LIN {X 0,Y 302.837,Z 619.691,A -85,B 0,C 180,E1 -24110.683,E2 -24110.683} C_VEL
LIN {X 0,Y 303.085,Z 619.66,A -85,B 0,C 180,E1 -24113.589,E2 -24113.589} C_VEL
LIN {X 0,Y 303.031,Z 619.668,A -85,B 0,C 180,E1 -24117.351,E2 -24117.351} C_VEL
LIN {X 0,Y 303.108,Z 619.662,A -85,B 0,C 180,E1 -24120,E2 -24120} C_VEL
LIN {X 0,Y 303.072,Z 619.665,A -85,B 0,C 180,E1 -24123.976,E2 -24123.976} C_VEL
LIN {X 0,Y 302.989,Z 619.674,A -85,B 0,C 180,E1 -24126.638,E2 -24126.638} C_VEL
LIN {X 0,Y 302.772,Z 619.699,A -85,B 0,C 180,E1 -24130.666,E2 -24130.666} C_VEL
LIN {X 0,Y 302.721,Z 619.706,A -85,B 0,C 180,E1 -24133.638,E2 -24133.638} C_VEL
LIN {X 0,Y 302.599,Z 619.723,A -85,B 0,C 180,E1 -24137.513,E2 -24137.513} C_VEL
LIN {X 0,Y 302.618,Z 619.72,A -85,B 0,C 180,E1 -24141.737,E2 -24141.737} C_VEL
LIN {X 0,Y 302.58,Z 619.729,A -85,B 0,C 180,E1 -24146.094,E2 -24146.094} C_VEL
LIN {X 0,Y 302.525,Z 619.73,A -85,B 0,C 180,E1 -24149.093,E2 -24149.093} C_VEL
LIN {X 0,Y 302.517,Z 619.734,A -85,B 0,C 180,E1 -24152.178,E2 -24152.178} C_VEL
LIN {X 0,Y 302.558,Z 619.731,A -85,B 0,C 180,E1 -24155.877,E2 -24155.877} C_VEL
LIN {X 0,Y 302.508,Z 619.732,A -85,B 0,C 180,E1 -24158.695,E2 -24158.695} C_VEL
LIN {X 0,Y 302.518,Z 619.734,A -85,B 0,C 180,E1 -24162.19,E2 -24162.19} C_VEL
LIN {X 0,Y 302.516,Z 619.736,A -85,B 0,C 180,E1 -24165.84,E2 -24165.84} C_VEL
LIN {X 0,Y 301.902,Z 619.818,A -85,B 0,C 180,E1 -24166.951,E2 -24166.951} C_VEL
LIN {X 0,Y 299.026,Z 620.17,A -85,B 0,C 180,E1 -24168.76,E2 -24168.76} C_VEL
LIN {X 0,Y 296.57,Z 620.472,A -85,B 0,C 180,E1 -24170.228,E2 -24170.228} C_VEL
LIN {X 0,Y 295.543,Z 620.598,A -85,B 0,C 180,E1 -24171.366,E2 -24171.366} C_VEL
LIN {X 0,Y 295.477,Z 620.608,A -85,B 0,C 180,E1 -24171.752,E2 -24171.752} C_VEL
LIN {X 0,Y 295.463,Z 620.611,A -85,B 0,C 180,E1 -24175.323,E2 -24175.323} C_VEL
LIN {X 0,Y 295.472,Z 620.609,A -85,B 0,C 180,E1 -24178.585,E2 -24178.585} C_VEL
LIN {X 0,Y 295.688,Z 620.648,A -85,B 0,C 180,E1 -24182.966,E2 -24182.966} C_VEL
LIN {X 0,Y 297.523,Z 631.227,A -85,B 0,C 180,E1 -24186.408,E2 -24186.408} C_VEL
LIN {X 0,Y 296.857,Z 636.884,A -85,B 0,C 180,E1 -24188.184,E2 -24188.184} C_VEL
LIN {X 0,Y 296.097,Z 642.614,A -85,B 0,C 180,E1 -24189.913,E2 -24189.913} C_VEL
LIN {X 0,Y 297.168,Z 664.042,A -85,B 0,C 180,E1 -24190.732,E2 -24190.732} C_VEL
LIN {X 0,Y 299.254,Z 687.174,A -85,B 0,C 180,E1 -24191.624,E2 -24191.624} C_VEL
LIN {X 0,Y 297.458,Z 748.577,A -85,B 0,C 180,E1 -24193.894,E2 -24193.894} C_VEL
LIN {X 0,Y 296.972,Z 759.313,A -85,B 0,C 180,E1 -24194.438,E2 -24194.438} C_VEL
LIN {X 0,Y 296.571,Z 769.561,A -85,B 0,C 180,E1 -24195.123,E2 -24195.123} C_VEL
LIN {X 0,Y 296.15,Z 779.319,A -85,B 0,C 180,E1 -24195.942,E2 -24195.942} C_VEL
LIN {X 0,Y 295.546,Z 789.452,A -85,B 0,C 180,E1 -24196.989,E2 -24196.989} C_VEL
LIN {X 0,Y 294.854,Z 798.937,A -85,B 0,C 180,E1 -24198.177,E2 -24198.177} C_VEL
LIN {X 0,Y 294.346,Z 806.961,A -85,B 0,C 180,E1 -24199.373,E2 -24199.373} C_VEL
LIN {X 0,Y 293.912,Z 814.791,A -85,B 0,C 180,E1 -24200.743,E2 -24200.743} C_VEL
LIN {X 0,Y 293.521,Z 822.971,A -85,B 0,C 180,E1 -24202.458,E2 -24202.458} C_VEL
LIN {X 0,Y 293.293,Z 829.787,A -85,B 0,C 180,E1 -24204.175,E2 -24204.175} C_VEL
LIN {X 0,Y 293.161,Z 835.457,A -85,B 0,C 180,E1 -24205.89,E2 -24205.89} C_VEL
LIN {X 0,Y 293.07,Z 839.33,A -85,B 0,C 180,E1 -24207.26,E2 -24207.26} C_VEL
LIN {X 0,Y 292.986,Z 843.949,A -85,B 0,C 180,E1 -24209.315,E2 -24209.315} C_VEL
LIN {X 0,Y 292.858,Z 847.401,A -85,B 0,C 180,E1 -24211.371,E2 -24211.371} C_VEL
LIN {X 0,Y 292.722,Z 850.314,A -85,B 0,C 180,E1 -24214.117,E2 -24214.117} C_VEL
LIN {X 0,Y 292.801,Z 851.206,A -85,B 0,C 180,E1 -24215.491,E2 -24215.491} C_VEL
LIN {X 0,Y 293.422,Z 851.753,A -85,B 0,C 180,E1 -24218.235,E2 -24218.235} C_VEL
LIN {X 0,Y 294.835,Z 850.611,A -85,B 0,C 180,E1 -24220.956,E2 -24220.956} C_VEL
LIN {X 0,Y 295.841,Z 849.532,A -85,B 0,C 180,E1 -24222.304,E2 -24222.304} C_VEL
LIN {X 0,Y 298.382,Z 846.007,A -85,B 0,C 180,E1 -24224.965,E2 -24224.965} C_VEL
LIN {X 0,Y 300.802,Z 842.241,A -85,B 0,C 180,E1 -24226.923,E2 -24226.923} C_VEL
LIN {X 0,Y 303.719,Z 836.954,A -85,B 0,C 180,E1 -24228.994,E2 -24228.994} C_VEL
LIN {X 0,Y 306.732,Z 831.292,A -85,B 0,C 180,E1 -24230.73,E2 -24230.73} C_VEL
LIN {X 0,Y 310.324,Z 823.881,A -85,B 0,C 180,E1 -24232.564,E2 -24232.564} C_VEL
LIN {X 0,Y 313.59,Z 816.478,A -85,B 0,C 180,E1 -24234.057,E2 -24234.057} C_VEL
LIN {X 0,Y 316.462,Z 809.57,A -85,B 0,C 180,E1 -24235.219,E2 -24235.219} C_VEL
LIN {X 0,Y 320.265,Z 799.204,A -85,B 0,C 180,E1 -24236.638,E2 -24236.638} C_VEL
LIN {X 0,Y 323.576,Z 789.286,A -85,B 0,C 180,E1 -24237.737,E2 -24237.737} C_VEL
LIN {X 0,Y 326.213,Z 780.533,A -85,B 0,C 180,E1 -24238.539,E2 -24238.539} C_VEL
LIN {X 0,Y 328.97,Z 769.976,A -85,B 0,C 180,E1 -24239.322,E2 -24239.322} C_VEL
LIN {X 0,Y 331.28,Z 759.343,A -85,B 0,C 180,E1 -24239.95,E2 -24239.95} C_VEL
LIN {X 0,Y 333.149,Z 748.652,A -85,B 0,C 180,E1 -24240.438,E2 -24240.438} C_VEL
LIN {X 0,Y 338.393,Z 705.295,A -85,B 0,C 180,E1 -24241.998,E2 -24241.998} C_VEL
LIN {X 0,Y 337.719,Z 697.125,A -85,B 0,C 180,E1 -24242.726,E2 -24242.726} C_VEL
LIN {X 0,Y 334.207,Z 688.297,A -85,B 0,C 180,E1 -24244.31,E2 -24244.31} C_VEL
LIN {X 0,Y 331.258,Z 682.06,A -85,B 0,C 180,E1 -24245.751,E2 -24245.751} C_VEL
LIN {X 0,Y 327.965,Z 675.305,A -85,B 0,C 180,E1 -24247.543,E2 -24247.543} C_VEL
LIN {X 0,Y 324.716,Z 669.541,A -85,B 0,C 180,E1 -24249.539,E2 -24249.539} C_VEL
LIN {X 0,Y 321.554,Z 664.083,A -85,B 0,C 180,E1 -24252.001,E2 -24252.001} C_VEL
LIN {X 0,Y 318.265,Z 658.7,A -85,B 0,C 180,E1 -24255.91,E2 -24255.91} C_VEL
LIN {X 0,Y 317.647,Z 657.399,A -85,B 0,C 180,E1 -24257.187,E2 -24257.187} C_VEL
LIN {X 0,Y 317.004,Z 656.38,A -85,B 0,C 180,E1 -24260.15,E2 -24260.15} C_VEL
LIN {X 0,Y 317.643,Z 656.7,A -85,B 0,C 180,E1 -24263.066,E2 -24263.066} C_VEL
LIN {X 0,Y 319.697,Z 659.747,A -85,B 0,C 180,E1 -24266.364,E2 -24266.364} C_VEL
LIN {X 0,Y 321.404,Z 661.42,A -85,B 0,C 180,E1 -24268.005,E2 -24268.005} C_VEL
LIN {X 0,Y 324.361,Z 665.767,A -85,B 0,C 180,E1 -24270.344,E2 -24270.344} C_VEL
LIN {X 0,Y 328.033,Z 671.683,A -85,B 0,C 180,E1 -24272.652,E2 -24272.652} C_VEL
LIN {X 0,Y 331.25,Z 677.099,A -85,B 0,C 180,E1 -24274.349,E2 -24274.349} C_VEL
LIN {X 0,Y 334.603,Z 683.345,A -85,B 0,C 180,E1 -24275.961,E2 -24275.961} C_VEL
LIN {X 0,Y 338.734,Z 692.186,A -85,B 0,C 180,E1 -24277.727,E2 -24277.727} C_VEL
LIN {X 0,Y 339.508,Z 694.26,A -85,B 0,C 180,E1 -24278.072,E2 -24278.072} C_VEL
LIN {X 0,Y 333.571,Z 740.577,A -85,B 0,C 180,E1 -24279.688,E2 -24279.688} C_VEL
LIN {X 0,Y 331.396,Z 753.38,A -85,B 0,C 180,E1 -24280.314,E2 -24280.314} C_VEL
LIN {X 0,Y 328.594,Z 766.328,A -85,B 0,C 180,E1 -24281.191,E2 -24281.191} C_VEL
LIN {X 0,Y 325.658,Z 777.244,A -85,B 0,C 180,E1 -24282.151,E2 -24282.151} C_VEL
LIN {X 0,Y 322.446,Z 787.5,A -85,B 0,C 180,E1 -24283.277,E2 -24283.277} C_VEL
LIN {X 0,Y 319.216,Z 796.785,A -85,B 0,C 180,E1 -24284.518,E2 -24284.518} C_VEL
LIN {X 0,Y 316.657,Z 803.539,A -85,B 0,C 180,E1 -24285.59,E2 -24285.59} C_VEL
LIN {X 0,Y 313.29,Z 811.378,A -85,B 0,C 180,E1 -24287.08,E2 -24287.08} C_VEL
LIN {X 0,Y 310.148,Z 817.968,A -85,B 0,C 180,E1 -24288.602,E2 -24288.602} C_VEL
LIN {X 0,Y 307.208,Z 823.519,A -85,B 0,C 180,E1 -24290.154,E2 -24290.154} C_VEL
LIN {X 0,Y 304.061,Z 828.963,A -85,B 0,C 180,E1 -24292.055,E2 -24292.055} C_VEL
LIN {X 0,Y 301.266,Z 833.24,A -85,B 0,C 180,E1 -24293.994,E2 -24293.994} C_VEL
LIN {X 0,Y 298.807,Z 836.453,A -85,B 0,C 180,E1 -24295.967,E2 -24295.967} C_VEL
LIN {X 0,Y 297.435,Z 838.026,A -85,B 0,C 180,E1 -24297.3,E2 -24297.3} C_VEL
LIN {X 0,Y 295.302,Z 839.94,A -85,B 0,C 180,E1 -24300,E2 -24300} C_VEL
LIN {X 0,Y 294.324,Z 840.259,A -85,B 0,C 180,E1 -24301.739,E2 -24301.739} C_VEL
LIN {X 0,Y 293.199,Z 839.49,A -85,B 0,C 180,E1 -24304.378,E2 -24304.378} C_VEL
LIN {X 0,Y 292.566,Z 837.401,A -85,B 0,C 180,E1 -24306.875,E2 -24306.875} C_VEL
LIN {X 0,Y 292.43,Z 834.605,A -85,B 0,C 180,E1 -24308.956,E2 -24308.956} C_VEL
LIN {X 0,Y 292.511,Z 830.698,A -85,B 0,C 180,E1 -24311.044,E2 -24311.044} C_VEL
LIN {X 0,Y 292.608,Z 825.536,A -85,B 0,C 180,E1 -24313.144,E2 -24313.144} C_VEL
LIN {X 0,Y 292.927,Z 820.251,A -85,B 0,C 180,E1 -24314.895,E2 -24314.895} C_VEL
LIN {X 0,Y 293.217,Z 813.79,A -85,B 0,C 180,E1 -24316.657,E2 -24316.657} C_VEL
LIN {X 0,Y 293.626,Z 805.948,A -85,B 0,C 180,E1 -24318.425,E2 -24318.425} C_VEL
LIN {X 0,Y 294.138,Z 797.477,A -85,B 0,C 180,E1 -24320.018,E2 -24320.018} C_VEL
LIN {X 0,Y 294.659,Z 788.683,A -85,B 0,C 180,E1 -24321.405,E2 -24321.405} C_VEL
LIN {X 0,Y 295.243,Z 779.055,A -85,B 0,C 180,E1 -24322.675,E2 -24322.675} C_VEL
LIN {X 0,Y 295.9,Z 769.478,A -85,B 0,C 180,E1 -24323.729,E2 -24323.729} C_VEL
LIN {X 0,Y 296.363,Z 759.6,A -85,B 0,C 180,E1 -24324.617,E2 -24324.617} C_VEL
LIN {X 0,Y 296.858,Z 748.44,A -85,B 0,C 180,E1 -24325.412,E2 -24325.412} C_VEL
LIN {X 0,Y 297.256,Z 737.936,A -85,B 0,C 180,E1 -24325.984,E2 -24325.984} C_VEL
LIN {X 0,Y 298.194,Z 711.392,A -85,B 0,C 180,E1 -24326.998,E2 -24326.998} C_VEL
LIN {X 0,Y 299.606,Z 662.208,A -85,B 0,C 180,E1 -24328.786,E2 -24328.786} C_VEL
LIN {X 0,Y 296.95,Z 636.125,A -85,B 0,C 180,E1 -24329.8,E2 -24329.8} C_VEL
LIN {X 0,Y 296.516,Z 629.06,A -85,B 0,C 180,E1 -24330.075,E2 -24330.075} C_VEL
LIN {X 0,Y 296.625,Z 625.432,A -85,B 0,C 180,E1 -24331.298,E2 -24331.298} C_VEL
LIN {X 0,Y 295.765,Z 620.573,A -85,B 0,C 180,E1 -24333.003,E2 -24333.003} C_VEL
LIN {X 0,Y 295.506,Z 620.608,A -85,B 0,C 180,E1 -24338.044,E2 -24338.044} C_VEL
LIN {X 0,Y 295.482,Z 620.61,A -85,B 0,C 180,E1 -24341.585,E2 -24341.585} C_VEL
LIN {X 0,Y 295.494,Z 620.605,A -85,B 0,C 180,E1 -24345.326,E2 -24345.326} C_VEL
LIN {X 0,Y 295.494,Z 620.607,A -85,B 0,C 180,E1 -24349.334,E2 -24349.334} C_VEL
LIN {X 0,Y 295.504,Z 620.61,A -85,B 0,C 180,E1 -24351.954,E2 -24351.954} C_VEL
LIN {X 0,Y 295.479,Z 620.61,A -85,B 0,C 180,E1 -24356.065,E2 -24356.065} C_VEL
LIN {X 0,Y 295.502,Z 620.61,A -85,B 0,C 180,E1 -24360.147,E2 -24360.147} C_VEL
LIN {X 0,Y 295.55,Z 620.6,A -85,B 0,C 180,E1 -24364.234,E2 -24364.234} C_VEL
LIN {X 0,Y 295.583,Z 620.596,A -85,B 0,C 180,E1 -24367.718,E2 -24367.718} C_VEL
LIN {X 0,Y 295.632,Z 620.593,A -85,B 0,C 180,E1 -24372.06,E2 -24372.06} C_VEL
LIN {X 0,Y 295.769,Z 620.573,A -85,B 0,C 180,E1 -24376.301,E2 -24376.301} C_VEL
LIN {X 0,Y 295.785,Z 620.572,A -85,B 0,C 180,E1 -24380.458,E2 -24380.458} C_VEL
LIN {X 0,Y 295.998,Z 620.545,A -85,B 0,C 180,E1 -24383.65,E2 -24383.65} C_VEL
LIN {X 0,Y 295.989,Z 620.544,A -85,B 0,C 180,E1 -24387.287,E2 -24387.287} C_VEL
LIN {X 0,Y 296.083,Z 620.539,A -85,B 0,C 180,E1 -24390,E2 -24390} C_VEL
LIN {X 0,Y 296.041,Z 620.539,A -85,B 0,C 180,E1 -24394.07,E2 -24394.07} C_VEL
LIN {X 0,Y 295.931,Z 620.551,A -85,B 0,C 180,E1 -24396.796,E2 -24396.796} C_VEL
LIN {X 0,Y 295.733,Z 620.577,A -85,B 0,C 180,E1 -24400.922,E2 -24400.922} C_VEL
LIN {X 0,Y 295.765,Z 620.575,A -85,B 0,C 180,E1 -24403.84,E2 -24403.84} C_VEL
LIN {X 0,Y 295.637,Z 620.59,A -85,B 0,C 180,E1 -24408.613,E2 -24408.613} C_VEL
LIN {X 0,Y 295.579,Z 620.596,A -85,B 0,C 180,E1 -24412.454,E2 -24412.454} C_VEL
LIN {X 0,Y 295.549,Z 620.6,A -85,B 0,C 180,E1 -24415.766,E2 -24415.766} C_VEL
LIN {X 0,Y 295.505,Z 620.609,A -85,B 0,C 180,E1 -24419.852,E2 -24419.852} C_VEL
LIN {X 0,Y 295.532,Z 620.603,A -85,B 0,C 180,E1 -24423.95,E2 -24423.95} C_VEL
LIN {X 0,Y 295.561,Z 620.604,A -85,B 0,C 180,E1 -24428.037,E2 -24428.037} C_VEL
LIN {X 0,Y 295.515,Z 620.605,A -85,B 0,C 180,E1 -24431.58,E2 -24431.58} C_VEL
LIN {X 0,Y 295.493,Z 620.605,A -85,B 0,C 180,E1 -24435.326,E2 -24435.326} C_VEL
LIN {X 0,Y 295.543,Z 620.601,A -85,B 0,C 180,E1 -24439.324,E2 -24439.324} C_VEL
LIN {X 0,Y 295.55,Z 620.599,A -85,B 0,C 180,E1 -24443.686,E2 -24443.686} C_VEL
LIN {X 0,Y 295.496,Z 620.606,A -85,B 0,C 180,E1 -24446.963,E2 -24446.963} C_VEL
LIN {X 0,Y 295.518,Z 620.603,A -85,B 0,C 180,E1 -24451.28,E2 -24451.28} C_VEL
LIN {X 0,Y 295.572,Z 620.596,A -85,B 0,C 180,E1 -24454.751,E2 -24454.751} C_VEL
LIN {X 0,Y 295.584,Z 620.598,A -85,B 0,C 180,E1 -24457.719,E2 -24457.719} C_VEL
LIN {X 0,Y 295.617,Z 620.592,A -85,B 0,C 180,E1 -24462.06,E2 -24462.06} C_VEL
LIN {X 0,Y 295.685,Z 620.586,A -85,B 0,C 180,E1 -24466.298,E2 -24466.298} C_VEL
LIN {X 0,Y 295.789,Z 620.57,A -85,B 0,C 180,E1 -24470.459,E2 -24470.459} C_VEL
LIN {X 0,Y 296.045,Z 620.536,A -85,B 0,C 180,E1 -24473.575,E2 -24473.575} C_VEL
LIN {X 0,Y 295.994,Z 620.545,A -85,B 0,C 180,E1 -24477.288,E2 -24477.288} C_VEL
LIN {X 0,Y 296.085,Z 620.537,A -85,B 0,C 180,E1 -24480,E2 -24480} C_VEL
LIN {X 0,Y 296.042,Z 620.542,A -85,B 0,C 180,E1 -24484.071,E2 -24484.071} C_VEL
LIN {X 0,Y 295.935,Z 620.552,A -85,B 0,C 180,E1 -24486.797,E2 -24486.797} C_VEL
LIN {X 0,Y 295.731,Z 620.575,A -85,B 0,C 180,E1 -24490.923,E2 -24490.923} C_VEL
LIN {X 0,Y 295.684,Z 620.584,A -85,B 0,C 180,E1 -24493.774,E2 -24493.774} C_VEL
LIN {X 0,Y 295.571,Z 620.602,A -85,B 0,C 180,E1 -24497.944,E2 -24497.944} C_VEL
LIN {X 0,Y 295.55,Z 620.6,A -85,B 0,C 180,E1 -24502.284,E2 -24502.284} C_VEL
LIN {X 0,Y 295.553,Z 620.602,A -85,B 0,C 180,E1 -24505.766,E2 -24505.766} C_VEL
LIN {X 0,Y 295.496,Z 620.61,A -85,B 0,C 180,E1 -24509.854,E2 -24509.854} C_VEL
LIN {X 0,Y 295.477,Z 620.612,A -85,B 0,C 180,E1 -24513.933,E2 -24513.933} C_VEL
LIN {X 0,Y 295.503,Z 620.608,A -85,B 0,C 180,E1 -24516.341,E2 -24516.341} C_VEL
LIN {X 0,Y 295.484,Z 620.605,A -85,B 0,C 180,E1 -24520.663,E2 -24520.663} C_VEL
LIN {X 0,Y 295.465,Z 620.611,A -85,B 0,C 180,E1 -24524.668,E2 -24524.668} C_VEL
LIN {X 0,Y 295.458,Z 620.612,A -85,B 0,C 180,E1 -24528.41,E2 -24528.41} C_VEL
LIN {X 0,Y 295.477,Z 620.608,A -85,B 0,C 180,E1 -24531.752,E2 -24531.752} C_VEL
LIN {X 0,Y 294.852,Z 620.693,A -85,B 0,C 180,E1 -24532.89,E2 -24532.89} C_VEL
LIN {X 0,Y 291.999,Z 621.053,A -85,B 0,C 180,E1 -24534.743,E2 -24534.743} C_VEL
LIN {X 0,Y 289.553,Z 621.354,A -85,B 0,C 180,E1 -24536.248,E2 -24536.248} C_VEL
LIN {X 0,Y 288.503,Z 621.481,A -85,B 0,C 180,E1 -24537.413,E2 -24537.413} C_VEL
LIN {X 0,Y 288.42,Z 621.49,A -85,B 0,C 180,E1 -24537.809,E2 -24537.809} C_VEL
LIN {X 0,Y 288.638,Z 621.459,A -85,B 0,C 180,E1 -24542.94,E2 -24542.94} C_VEL
LIN {X 0,Y 290.454,Z 631.8,A -85,B 0,C 180,E1 -24546.404,E2 -24546.404} C_VEL
LIN {X 0,Y 289.16,Z 641.261,A -85,B 0,C 180,E1 -24549.437,E2 -24549.437} C_VEL
LIN {X 0,Y 289.032,Z 642.243,A -85,B 0,C 180,E1 -24549.752,E2 -24549.752} C_VEL
LIN {X 0,Y 289.981,Z 663.201,A -85,B 0,C 180,E1 -24550.584,E2 -24550.584} C_VEL
LIN {X 0,Y 292.153,Z 688.015,A -85,B 0,C 180,E1 -24551.564,E2 -24551.564} C_VEL
LIN {X 0,Y 290.378,Z 748.001,A -85,B 0,C 180,E1 -24553.85,E2 -24553.85} C_VEL
LIN {X 0,Y 289.894,Z 758.725,A -85,B 0,C 180,E1 -24554.407,E2 -24554.407} C_VEL
LIN {X 0,Y 289.471,Z 769.557,A -85,B 0,C 180,E1 -24555.156,E2 -24555.156} C_VEL
LIN {X 0,Y 289.056,Z 779.032,A -85,B 0,C 180,E1 -24555.977,E2 -24555.977} C_VEL
LIN {X 0,Y 288.48,Z 788.884,A -85,B 0,C 180,E1 -24557.021,E2 -24557.021} C_VEL
LIN {X 0,Y 287.809,Z 798.375,A -85,B 0,C 180,E1 -24558.24,E2 -24558.24} C_VEL
LIN {X 0,Y 287.243,Z 807.477,A -85,B 0,C 180,E1 -24559.64,E2 -24559.64} C_VEL
LIN {X 0,Y 286.871,Z 814.339,A -85,B 0,C 180,E1 -24560.868,E2 -24560.868} C_VEL
LIN {X 0,Y 286.468,Z 822.558,A -85,B 0,C 180,E1 -24562.625,E2 -24562.625} C_VEL
LIN {X 0,Y 286.245,Z 829.414,A -85,B 0,C 180,E1 -24564.383,E2 -24564.383} C_VEL
LIN {X 0,Y 286.132,Z 834.135,A -85,B 0,C 180,E1 -24565.789,E2 -24565.789} C_VEL
LIN {X 0,Y 286.057,Z 839.841,A -85,B 0,C 180,E1 -24567.895,E2 -24567.895} C_VEL
LIN {X 0,Y 285.878,Z 844.259,A -85,B 0,C 180,E1 -24570,E2 -24570} C_VEL
LIN {X 0,Y 285.814,Z 846.53,A -85,B 0,C 180,E1 -24571.405,E2 -24571.405} C_VEL
LIN {X 0,Y 285.66,Z 849.809,A -85,B 0,C 180,E1 -24574.219,E2 -24574.219} C_VEL
LIN {X 0,Y 286.003,Z 851.316,A -85,B 0,C 180,E1 -24577.034,E2 -24577.034} C_VEL
LIN {X 0,Y 286.388,Z 851.552,A -85,B 0,C 180,E1 -24578.439,E2 -24578.439} C_VEL
LIN {X 0,Y 287.881,Z 850.761,A -85,B 0,C 180,E1 -24581.224,E2 -24581.224} C_VEL
LIN {X 0,Y 290.081,Z 848.305,A -85,B 0,C 180,E1 -24583.973,E2 -24583.973} C_VEL
LIN {X 0,Y 292.352,Z 845.43,A -85,B 0,C 180,E1 -24585.994,E2 -24585.994} C_VEL
LIN {X 0,Y 294.977,Z 841.54,A -85,B 0,C 180,E1 -24587.981,E2 -24587.981} C_VEL
LIN {X 0,Y 297.915,Z 836.629,A -85,B 0,C 180,E1 -24589.932,E2 -24589.932} C_VEL
LIN {X 0,Y 301.46,Z 830.469,A -85,B 0,C 180,E1 -24591.825,E2 -24591.825} C_VEL
LIN {X 0,Y 304.579,Z 824.334,A -85,B 0,C 180,E1 -24593.372,E2 -24593.372} C_VEL
LIN {X 0,Y 308.026,Z 817.016,A -85,B 0,C 180,E1 -24594.878,E2 -24594.878} C_VEL
LIN {X 0,Y 311.797,Z 808.331,A -85,B 0,C 180,E1 -24596.339,E2 -24596.339} C_VEL
LIN {X 0,Y 315.433,Z 799.076,A -85,B 0,C 180,E1 -24597.616,E2 -24597.616} C_VEL
LIN {X 0,Y 318.458,Z 790.595,A -85,B 0,C 180,E1 -24598.581,E2 -24598.581} C_VEL
LIN {X 0,Y 321.646,Z 780.472,A -85,B 0,C 180,E1 -24599.519,E2 -24599.519} C_VEL
LIN {X 0,Y 324.426,Z 770.299,A -85,B 0,C 180,E1 -24600.275,E2 -24600.275} C_VEL
LIN {X 0,Y 326.942,Z 759.074,A -85,B 0,C 180,E1 -24600.943,E2 -24600.943} C_VEL
LIN {X 0,Y 329.084,Z 747.192,A -85,B 0,C 180,E1 -24601.483,E2 -24601.483} C_VEL
LIN {X 0,Y 334.275,Z 707.304,A -85,B 0,C 180,E1 -24602.933,E2 -24602.933} C_VEL
LIN {X 0,Y 333.772,Z 701.007,A -85,B 0,C 180,E1 -24603.513,E2 -24603.513} C_VEL
LIN {X 0,Y 330.79,Z 693.264,A -85,B 0,C 180,E1 -24604.981,E2 -24604.981} C_VEL
LIN {X 0,Y 327.454,Z 685.862,A -85,B 0,C 180,E1 -24606.725,E2 -24606.725} C_VEL
LIN {X 0,Y 324.892,Z 680.702,A -85,B 0,C 180,E1 -24608.26,E2 -24608.26} C_VEL
LIN {X 0,Y 322.437,Z 675.951,A -85,B 0,C 180,E1 -24609.91,E2 -24609.91} C_VEL
LIN {X 0,Y 319.428,Z 670.551,A -85,B 0,C 180,E1 -24612.396,E2 -24612.396} C_VEL
LIN {X 0,Y 316.533,Z 665.443,A -85,B 0,C 180,E1 -24616.15,E2 -24616.15} C_VEL
LIN {X 0,Y 315.891,Z 664.114,A -85,B 0,C 180,E1 -24617.581,E2 -24617.581} C_VEL
LIN {X 0,Y 315.454,Z 663.32,A -85,B 0,C 180,E1 -24619.915,E2 -24619.915} C_VEL
LIN {X 0,Y 315.998,Z 663.564,A -85,B 0,C 180,E1 -24622.938,E2 -24622.938} C_VEL
LIN {X 0,Y 318.407,Z 667.025,A -85,B 0,C 180,E1 -24626.714,E2 -24626.714} C_VEL
LIN {X 0,Y 319.491,Z 668.209,A -85,B 0,C 180,E1 -24627.785,E2 -24627.785} C_VEL
LIN {X 0,Y 322.258,Z 672.384,A -85,B 0,C 180,E1 -24630.072,E2 -24630.072} C_VEL
LIN {X 0,Y 325.516,Z 677.906,A -85,B 0,C 180,E1 -24632.239,E2 -24632.239} C_VEL
LIN {X 0,Y 328.487,Z 683.176,A -85,B 0,C 180,E1 -24633.929,E2 -24633.929} C_VEL
LIN {X 0,Y 331.907,Z 689.852,A -85,B 0,C 180,E1 -24635.628,E2 -24635.628} C_VEL
LIN {X 0,Y 335.207,Z 697.325,A -85,B 0,C 180,E1 -24637.145,E2 -24637.145} C_VEL
LIN {X 0,Y 329.42,Z 740.445,A -85,B 0,C 180,E1 -24638.687,E2 -24638.687} C_VEL
LIN {X 0,Y 327.35,Z 751.948,A -85,B 0,C 180,E1 -24639.243,E2 -24639.243} C_VEL
LIN {X 0,Y 324.379,Z 765.441,A -85,B 0,C 180,E1 -24640.117,E2 -24640.117} C_VEL
LIN {X 0,Y 320.915,Z 777.933,A -85,B 0,C 180,E1 -24641.219,E2 -24641.219} C_VEL
LIN {X 0,Y 317.751,Z 787.575,A -85,B 0,C 180,E1 -24642.274,E2 -24642.274} C_VEL
LIN {X 0,Y 314.681,Z 796.017,A -85,B 0,C 180,E1 -24643.406,E2 -24643.406} C_VEL
LIN {X 0,Y 311.446,Z 803.932,A -85,B 0,C 180,E1 -24644.677,E2 -24644.677} C_VEL
LIN {X 0,Y 307.904,Z 811.732,A -85,B 0,C 180,E1 -24646.18,E2 -24646.18} C_VEL
LIN {X 0,Y 304.585,Z 818.323,A -85,B 0,C 180,E1 -24647.718,E2 -24647.718} C_VEL
LIN {X 0,Y 301.45,Z 823.878,A -85,B 0,C 180,E1 -24649.287,E2 -24649.287} C_VEL
LIN {X 0,Y 297.979,Z 829.432,A -85,B 0,C 180,E1 -24651.298,E2 -24651.298} C_VEL
LIN {X 0,Y 295.128,Z 833.475,A -85,B 0,C 180,E1 -24653.184,E2 -24653.184} C_VEL
LIN {X 0,Y 293.337,Z 835.766,A -85,B 0,C 180,E1 -24654.519,E2 -24654.519} C_VEL
LIN {X 0,Y 290.324,Z 838.893,A -85,B 0,C 180,E1 -24657.234,E2 -24657.234} C_VEL
LIN {X 0,Y 289.181,Z 839.788,A -85,B 0,C 180,E1 -24658.612,E2 -24658.612} C_VEL
LIN {X 0,Y 287.29,Z 840.469,A -85,B 0,C 180,E1 -24661.554,E2 -24661.554} C_VEL
LIN {X 0,Y 286.143,Z 839.382,A -85,B 0,C 180,E1 -24664.279,E2 -24664.279} C_VEL
LIN {X 0,Y 285.738,Z 838.347,A -85,B 0,C 180,E1 -24665.627,E2 -24665.627} C_VEL
LIN {X 0,Y 285.372,Z 834.816,A -85,B 0,C 180,E1 -24668.468,E2 -24668.468} C_VEL
LIN {X 0,Y 285.468,Z 830.661,A -85,B 0,C 180,E1 -24670.744,E2 -24670.744} C_VEL
LIN {X 0,Y 285.505,Z 825.885,A -85,B 0,C 180,E1 -24672.756,E2 -24672.756} C_VEL
LIN {X 0,Y 285.88,Z 819.397,A -85,B 0,C 180,E1 -24674.907,E2 -24674.907} C_VEL
LIN {X 0,Y 286.195,Z 812.733,A -85,B 0,C 180,E1 -24676.712,E2 -24676.712} C_VEL
LIN {X 0,Y 286.516,Z 806.287,A -85,B 0,C 180,E1 -24678.193,E2 -24678.193} C_VEL
LIN {X 0,Y 287.082,Z 796.971,A -85,B 0,C 180,E1 -24679.973,E2 -24679.973} C_VEL
LIN {X 0,Y 287.534,Z 789.089,A -85,B 0,C 180,E1 -24681.245,E2 -24681.245} C_VEL
LIN {X 0,Y 288.106,Z 779.872,A -85,B 0,C 180,E1 -24682.502,E2 -24682.502} C_VEL
LIN {X 0,Y 288.743,Z 770.306,A -85,B 0,C 180,E1 -24683.594,E2 -24683.594} C_VEL
LIN {X 0,Y 289.263,Z 759.549,A -85,B 0,C 180,E1 -24684.594,E2 -24684.594} C_VEL
LIN {X 0,Y 289.77,Z 749.256,A -85,B 0,C 180,E1 -24685.359,E2 -24685.359} C_VEL
LIN {X 0,Y 290.13,Z 738.33,A -85,B 0,C 180,E1 -24685.983,E2 -24685.983} C_VEL
LIN {X 0,Y 291.073,Z 712.412,A -85,B 0,C 180,E1 -24687.022,E2 -24687.022} C_VEL
LIN {X 0,Y 292.495,Z 662.407,A -85,B 0,C 180,E1 -24688.896,E2 -24688.896} C_VEL
LIN {X 0,Y 289.929,Z 637.285,A -85,B 0,C 180,E1 -24689.896,E2 -24689.896} C_VEL
LIN {X 0,Y 289.479,Z 629.205,A -85,B 0,C 180,E1 -24690.219,E2 -24690.219} C_VEL
LIN {X 0,Y 289.567,Z 626.185,A -85,B 0,C 180,E1 -24691.258,E2 -24691.258} C_VEL
LIN {X 0,Y 288.739,Z 621.448,A -85,B 0,C 180,E1 -24692.976,E2 -24692.976} C_VEL
LIN {X 0,Y 288.461,Z 621.48,A -85,B 0,C 180,E1 -24697.376,E2 -24697.376} C_VEL
LIN {X 0,Y 288.434,Z 621.486,A -85,B 0,C 180,E1 -24701.165,E2 -24701.165} C_VEL
LIN {X 0,Y 288.47,Z 621.48,A -85,B 0,C 180,E1 -24705.238,E2 -24705.238} C_VEL
LIN {X 0,Y 288.44,Z 621.485,A -85,B 0,C 180,E1 -24709.03,E2 -24709.03} C_VEL
LIN {X 0,Y 288.453,Z 621.484,A -85,B 0,C 180,E1 -24713.256,E2 -24713.256} C_VEL
LIN {X 0,Y 288.442,Z 621.486,A -85,B 0,C 180,E1 -24716.046,E2 -24716.046} C_VEL
LIN {X 0,Y 288.453,Z 621.484,A -85,B 0,C 180,E1 -24719.34,E2 -24719.34} C_VEL
LIN {X 0,Y 288.479,Z 621.481,A -85,B 0,C 180,E1 -24722.527,E2 -24722.527} C_VEL
LIN {X 0,Y 288.481,Z 621.479,A -85,B 0,C 180,E1 -24725.621,E2 -24725.621} C_VEL
LIN {X 0,Y 288.506,Z 621.478,A -85,B 0,C 180,E1 -24728.643,E2 -24728.643} C_VEL
LIN {X 0,Y 288.598,Z 621.468,A -85,B 0,C 180,E1 -24731.608,E2 -24731.608} C_VEL
LIN {X 0,Y 288.717,Z 621.452,A -85,B 0,C 180,E1 -24736.027,E2 -24736.027} C_VEL
LIN {X 0,Y 288.736,Z 621.452,A -85,B 0,C 180,E1 -24740.223,E2 -24740.223} C_VEL
LIN {X 0,Y 288.907,Z 621.425,A -85,B 0,C 180,E1 -24744.435,E2 -24744.435} C_VEL
LIN {X 0,Y 288.954,Z 621.42,A -85,B 0,C 180,E1 -24747.221,E2 -24747.221} C_VEL
LIN {X 0,Y 289.061,Z 621.413,A -85,B 0,C 180,E1 -24750,E2 -24750} C_VEL
LIN {X 0,Y 288.99,Z 621.417,A -85,B 0,C 180,E1 -24754.17,E2 -24754.17} C_VEL
LIN {X 0,Y 288.874,Z 621.43,A -85,B 0,C 180,E1 -24756.963,E2 -24756.963} C_VEL
LIN {X 0,Y 288.674,Z 621.456,A -85,B 0,C 180,E1 -24761.193,E2 -24761.193} C_VEL
LIN {X 0,Y 288.7,Z 621.454,A -85,B 0,C 180,E1 -24764.041,E2 -24764.041} C_VEL
LIN {X 0,Y 288.587,Z 621.467,A -85,B 0,C 180,E1 -24768.813,E2 -24768.813} C_VEL
LIN {X 0,Y 288.509,Z 621.475,A -85,B 0,C 180,E1 -24772.858,E2 -24772.858} C_VEL
LIN {X 0,Y 288.494,Z 621.482,A -85,B 0,C 180,E1 -24776.062,E2 -24776.062} C_VEL
LIN {X 0,Y 288.462,Z 621.483,A -85,B 0,C 180,E1 -24780.658,E2 -24780.658} C_VEL
LIN {X 0,Y 288.484,Z 621.479,A -85,B 0,C 180,E1 -24784.359,E2 -24784.359} C_VEL
LIN {X 0,Y 288.499,Z 621.478,A -85,B 0,C 180,E1 -24787.371,E2 -24787.371} C_VEL
LIN {X 0,Y 288.475,Z 621.481,A -85,B 0,C 180,E1 -24791.175,E2 -24791.175} C_VEL
LIN {X 0,Y 288.469,Z 621.48,A -85,B 0,C 180,E1 -24795.239,E2 -24795.239} C_VEL
LIN {X 0,Y 288.481,Z 621.48,A -85,B 0,C 180,E1 -24799.038,E2 -24799.038} C_VEL
LIN {X 0,Y 288.484,Z 621.477,A -85,B 0,C 180,E1 -24802.628,E2 -24802.628} C_VEL
LIN {X 0,Y 288.449,Z 621.488,A -85,B 0,C 180,E1 -24806.048,E2 -24806.048} C_VEL
LIN {X 0,Y 288.453,Z 621.484,A -85,B 0,C 180,E1 -24809.341,E2 -24809.341} C_VEL
LIN {X 0,Y 288.48,Z 621.478,A -85,B 0,C 180,E1 -24812.528,E2 -24812.528} C_VEL
LIN {X 0,Y 288.482,Z 621.481,A -85,B 0,C 180,E1 -24815.622,E2 -24815.622} C_VEL
LIN {X 0,Y 288.507,Z 621.478,A -85,B 0,C 180,E1 -24818.644,E2 -24818.644} C_VEL
LIN {X 0,Y 288.57,Z 621.47,A -85,B 0,C 180,E1 -24821.607,E2 -24821.607} C_VEL
LIN {X 0,Y 288.644,Z 621.464,A -85,B 0,C 180,E1 -24826.088,E2 -24826.088} C_VEL
LIN {X 0,Y 288.738,Z 621.45,A -85,B 0,C 180,E1 -24830.224,E2 -24830.224} C_VEL
LIN {X 0,Y 288.996,Z 621.414,A -85,B 0,C 180,E1 -24833.577,E2 -24833.577} C_VEL
LIN {X 0,Y 288.959,Z 621.421,A -85,B 0,C 180,E1 -24837.222,E2 -24837.222} C_VEL
LIN {X 0,Y 289.063,Z 621.411,A -85,B 0,C 180,E1 -24840,E2 -24840} C_VEL
LIN {X 0,Y 288.991,Z 621.42,A -85,B 0,C 180,E1 -24844.17,E2 -24844.17} C_VEL
LIN {X 0,Y 288.878,Z 621.431,A -85,B 0,C 180,E1 -24846.964,E2 -24846.964} C_VEL
LIN {X 0,Y 288.668,Z 621.455,A -85,B 0,C 180,E1 -24851.194,E2 -24851.194} C_VEL
LIN {X 0,Y 288.615,Z 621.467,A -85,B 0,C 180,E1 -24854.046,E2 -24854.046} C_VEL
LIN {X 0,Y 288.51,Z 621.476,A -85,B 0,C 180,E1 -24858.766,E2 -24858.766} C_VEL
LIN {X 0,Y 288.494,Z 621.476,A -85,B 0,C 180,E1 -24862.86,E2 -24862.86} C_VEL
LIN {X 0,Y 288.498,Z 621.483,A -85,B 0,C 180,E1 -24866.062,E2 -24866.062} C_VEL
LIN {X 0,Y 288.46,Z 621.482,A -85,B 0,C 180,E1 -24869.055,E2 -24869.055} C_VEL
LIN {X 0,Y 288.423,Z 621.488,A -85,B 0,C 180,E1 -24872.295,E2 -24872.295} C_VEL
LIN {X 0,Y 288.417,Z 621.49,A -85,B 0,C 180,E1 -24875.652,E2 -24875.652} C_VEL
LIN {X 0,Y 288.423,Z 621.487,A -85,B 0,C 180,E1 -24879.155,E2 -24879.155} C_VEL
LIN {X 0,Y 288.393,Z 621.49,A -85,B 0,C 180,E1 -24883.228,E2 -24883.228} C_VEL
LIN {X 0,Y 288.394,Z 621.491,A -85,B 0,C 180,E1 -24887.152,E2 -24887.152} C_VEL
LIN {X 0,Y 288.424,Z 621.483,A -85,B 0,C 180,E1 -24890.999,E2 -24890.999} C_VEL
LIN {X 0,Y 288.414,Z 621.491,A -85,B 0,C 180,E1 -24894.348,E2 -24894.348} C_VEL
LIN {X 0,Y 288.42,Z 621.49,A -85,B 0,C 180,E1 -24897.809,E2 -24897.809} C_VEL
LIN {X 0,Y 287.741,Z 621.574,A -85,B 0,C 180,E1 -24898.586,E2 -24898.586} C_VEL
LIN {X 0,Y 284.899,Z 621.929,A -85,B 0,C 180,E1 -24899.807,E2 -24899.807} C_VEL
LIN {X 0,Y 282.085,Z 622.278,A -85,B 0,C 180,E1 -24901.051,E2 -24901.051} C_VEL
LIN {X 0,Y 281.477,Z 622.352,A -85,B 0,C 180,E1 -24901.854,E2 -24901.854} C_VEL
LIN {X 0,Y 281.595,Z 622.38,A -85,B 0,C 180,E1 -24903.003,E2 -24903.003} C_VEL
LIN {X 0,Y 283.284,Z 631.691,A -85,B 0,C 180,E1 -24906.186,E2 -24906.186} C_VEL
LIN {X 0,Y 282.978,Z 635.472,A -85,B 0,C 180,E1 -24907.439,E2 -24907.439} C_VEL
LIN {X 0,Y 281.996,Z 642.055,A -85,B 0,C 180,E1 -24909.603,E2 -24909.603} C_VEL
LIN {X 0,Y 282.666,Z 659.547,A -85,B 0,C 180,E1 -24910.329,E2 -24910.329} C_VEL
LIN {X 0,Y 285.05,Z 688.721,A -85,B 0,C 180,E1 -24911.51,E2 -24911.51} C_VEL
LIN {X 0,Y 283.266,Z 748.576,A -85,B 0,C 180,E1 -24913.895,E2 -24913.895} C_VEL
LIN {X 0,Y 282.798,Z 759.092,A -85,B 0,C 180,E1 -24914.467,E2 -24914.467} C_VEL
LIN {X 0,Y 282.388,Z 769.13,A -85,B 0,C 180,E1 -24915.18,E2 -24915.18} C_VEL
LIN {X 0,Y 281.984,Z 778.814,A -85,B 0,C 180,E1 -24916.038,E2 -24916.038} C_VEL
LIN {X 0,Y 281.412,Z 788.231,A -85,B 0,C 180,E1 -24917.055,E2 -24917.055} C_VEL
LIN {X 0,Y 280.756,Z 797.804,A -85,B 0,C 180,E1 -24918.305,E2 -24918.305} C_VEL
LIN {X 0,Y 280.18,Z 806.964,A -85,B 0,C 180,E1 -24919.74,E2 -24919.74} C_VEL
LIN {X 0,Y 279.804,Z 813.878,A -85,B 0,C 180,E1 -24920.999,E2 -24920.999} C_VEL
LIN {X 0,Y 279.434,Z 822.151,A -85,B 0,C 180,E1 -24922.8,E2 -24922.8} C_VEL
LIN {X 0,Y 279.219,Z 829.048,A -85,B 0,C 180,E1 -24924.602,E2 -24924.602} C_VEL
LIN {X 0,Y 279.061,Z 834.759,A -85,B 0,C 180,E1 -24926.403,E2 -24926.403} C_VEL
LIN {X 0,Y 279.039,Z 838.619,A -85,B 0,C 180,E1 -24927.842,E2 -24927.842} C_VEL
LIN {X 0,Y 278.847,Z 843.245,A -85,B 0,C 180,E1 -24930,E2 -24930} C_VEL
LIN {X 0,Y 278.687,Z 846.718,A -85,B 0,C 180,E1 -24932.161,E2 -24932.161} C_VEL
LIN {X 0,Y 278.622,Z 849.158,A -85,B 0,C 180,E1 -24934.326,E2 -24934.326} C_VEL
LIN {X 0,Y 278.943,Z 851.027,A -85,B 0,C 180,E1 -24937.213,E2 -24937.213} C_VEL
LIN {X 0,Y 280.039,Z 851.21,A -85,B 0,C 180,E1 -24940.084,E2 -24940.084} C_VEL
LIN {X 0,Y 280.919,Z 850.792,A -85,B 0,C 180,E1 -24941.506,E2 -24941.506} C_VEL
LIN {X 0,Y 283.208,Z 848.701,A -85,B 0,C 180,E1 -24944.32,E2 -24944.32} C_VEL
LIN {X 0,Y 285.556,Z 846.055,A -85,B 0,C 180,E1 -24946.385,E2 -24946.385} C_VEL
LIN {X 0,Y 288.289,Z 842.457,A -85,B 0,C 180,E1 -24948.413,E2 -24948.413} C_VEL
LIN {X 0,Y 291.341,Z 837.822,A -85,B 0,C 180,E1 -24950.402,E2 -24950.402} C_VEL
LIN {X 0,Y 295.636,Z 830.83,A -85,B 0,C 180,E1 -24952.645,E2 -24952.645} C_VEL
LIN {X 0,Y 299.635,Z 823.422,A -85,B 0,C 180,E1 -24954.515,E2 -24954.515} C_VEL
LIN {X 0,Y 303.305,Z 816.088,A -85,B 0,C 180,E1 -24956.026,E2 -24956.026} C_VEL
LIN {X 0,Y 307.339,Z 807.293,A -85,B 0,C 180,E1 -24957.485,E2 -24957.485} C_VEL
LIN {X 0,Y 310.705,Z 799.021,A -85,B 0,C 180,E1 -24958.624,E2 -24958.624} C_VEL
LIN {X 0,Y 313.915,Z 790.391,A -85,B 0,C 180,E1 -24959.601,E2 -24959.601} C_VEL
LIN {X 0,Y 317.671,Z 778.904,A -85,B 0,C 180,E1 -24960.657,E2 -24960.657} C_VEL
LIN {X 0,Y 320.446,Z 769.133,A -85,B 0,C 180,E1 -24961.376,E2 -24961.376} C_VEL
LIN {X 0,Y 322.937,Z 758.501,A -85,B 0,C 180,E1 -24962.01,E2 -24962.01} C_VEL
LIN {X 0,Y 325.151,Z 746.824,A -85,B 0,C 180,E1 -24962.532,E2 -24962.532} C_VEL
LIN {X 0,Y 330.237,Z 709.104,A -85,B 0,C 180,E1 -24963.909,E2 -24963.909} C_VEL
LIN {X 0,Y 329.945,Z 705.124,A -85,B 0,C 180,E1 -24964.294,E2 -24964.294} C_VEL
LIN {X 0,Y 327.194,Z 697.653,A -85,B 0,C 180,E1 -24965.795,E2 -24965.795} C_VEL
LIN {X 0,Y 324.297,Z 690.968,A -85,B 0,C 180,E1 -24967.462,E2 -24967.462} C_VEL
LIN {X 0,Y 322.225,Z 686.611,A -85,B 0,C 180,E1 -24968.779,E2 -24968.779} C_VEL
LIN {X 0,Y 320.031,Z 682.101,A -85,B 0,C 180,E1 -24970.396,E2 -24970.396} C_VEL
LIN {X 0,Y 317.498,Z 677.227,A -85,B 0,C 180,E1 -24972.642,E2 -24972.642} C_VEL
LIN {X 0,Y 314.811,Z 672.291,A -85,B 0,C 180,E1 -24976.294,E2 -24976.294} C_VEL
LIN {X 0,Y 314.238,Z 670.995,A -85,B 0,C 180,E1 -24977.684,E2 -24977.684} C_VEL
LIN {X 0,Y 313.86,Z 670.296,A -85,B 0,C 180,E1 -24979.669,E2 -24979.669} C_VEL
LIN {X 0,Y 314.324,Z 670.351,A -85,B 0,C 180,E1 -24982.707,E2 -24982.707} C_VEL
LIN {X 0,Y 315.93,Z 673.13,A -85,B 0,C 180,E1 -24985.839,E2 -24985.839} C_VEL
LIN {X 0,Y 317.591,Z 674.959,A -85,B 0,C 180,E1 -24987.562,E2 -24987.562} C_VEL
LIN {X 0,Y 320.525,Z 679.73,A -85,B 0,C 180,E1 -24990.094,E2 -24990.094} C_VEL
LIN {X 0,Y 323.21,Z 684.528,A -85,B 0,C 180,E1 -24991.955,E2 -24991.955} C_VEL
LIN {X 0,Y 325.659,Z 689.033,A -85,B 0,C 180,E1 -24993.427,E2 -24993.427} C_VEL
LIN {X 0,Y 328.726,Z 695.182,A -85,B 0,C 180,E1 -24995.037,E2 -24995.037} C_VEL
LIN {X 0,Y 331.027,Z 701.045,A -85,B 0,C 180,E1 -24996.252,E2 -24996.252} C_VEL
LIN {X 0,Y 325.48,Z 740.542,A -85,B 0,C 180,E1 -24997.652,E2 -24997.652} C_VEL
LIN {X 0,Y 323.323,Z 752.102,A -85,B 0,C 180,E1 -24998.206,E2 -24998.206} C_VEL
LIN {X 0,Y 320.362,Z 764.756,A -85,B 0,C 180,E1 -24999.021,E2 -24999.021} C_VEL
LIN {X 0,Y 316.7,Z 777.379,A -85,B 0,C 180,E1 -25000.12,E2 -25000.12} C_VEL
LIN {X 0,Y 313.199,Z 787.63,A -85,B 0,C 180,E1 -25001.247,E2 -25001.247} C_VEL
LIN {X 0,Y 309.947,Z 796.138,A -85,B 0,C 180,E1 -25002.378,E2 -25002.378} C_VEL
LIN {X 0,Y 306.329,Z 804.564,A -85,B 0,C 180,E1 -25003.742,E2 -25003.742} C_VEL
LIN {X 0,Y 302.618,Z 812.216,A -85,B 0,C 180,E1 -25005.249,E2 -25005.249} C_VEL
LIN {X 0,Y 299.084,Z 818.702,A -85,B 0,C 180,E1 -25006.8,E2 -25006.8} C_VEL
LIN {X 0,Y 295.805,Z 824.223,A -85,B 0,C 180,E1 -25008.388,E2 -25008.388} C_VEL
LIN {X 0,Y 292.22,Z 829.591,A -85,B 0,C 180,E1 -25010.34,E2 -25010.34} C_VEL
LIN {X 0,Y 289.05,Z 833.787,A -85,B 0,C 180,E1 -25012.34,E2 -25012.34} C_VEL
LIN {X 0,Y 286.251,Z 836.935,A -85,B 0,C 180,E1 -25014.383,E2 -25014.383} C_VEL
LIN {X 0,Y 284.634,Z 838.506,A -85,B 0,C 180,E1 -25015.766,E2 -25015.766} C_VEL
LIN {X 0,Y 282.068,Z 840.37,A -85,B 0,C 180,E1 -25018.577,E2 -25018.577} C_VEL
LIN {X 0,Y 280.228,Z 840.511,A -85,B 0,C 180,E1 -25021.432,E2 -25021.432} C_VEL
LIN {X 0,Y 279.535,Z 840.088,A -85,B 0,C 180,E1 -25022.872,E2 -25022.872} C_VEL
LIN {X 0,Y 278.626,Z 837.82,A -85,B 0,C 180,E1 -25025.771,E2 -25025.771} C_VEL
LIN {X 0,Y 278.315,Z 835.022,A -85,B 0,C 180,E1 -25027.956,E2 -25027.956} C_VEL
LIN {X 0,Y 278.343,Z 831.181,A -85,B 0,C 180,E1 -25030.145,E2 -25030.145} C_VEL
LIN {X 0,Y 278.417,Z 826.118,A -85,B 0,C 180,E1 -25032.347,E2 -25032.347} C_VEL
LIN {X 0,Y 278.762,Z 819.714,A -85,B 0,C 180,E1 -25034.552,E2 -25034.552} C_VEL
LIN {X 0,Y 279.106,Z 813.164,A -85,B 0,C 180,E1 -25036.399,E2 -25036.399} C_VEL
LIN {X 0,Y 279.379,Z 807.113,A -85,B 0,C 180,E1 -25037.847,E2 -25037.847} C_VEL
LIN {X 0,Y 279.961,Z 797.526,A -85,B 0,C 180,E1 -25039.74,E2 -25039.74} C_VEL
LIN {X 0,Y 280.476,Z 788.447,A -85,B 0,C 180,E1 -25041.23,E2 -25041.23} C_VEL
LIN {X 0,Y 280.991,Z 779.902,A -85,B 0,C 180,E1 -25042.417,E2 -25042.417} C_VEL
LIN {X 0,Y 281.706,Z 769.317,A -85,B 0,C 180,E1 -25043.636,E2 -25043.636} C_VEL
LIN {X 0,Y 282.166,Z 759.414,A -85,B 0,C 180,E1 -25044.569,E2 -25044.569} C_VEL
LIN {X 0,Y 282.672,Z 749.048,A -85,B 0,C 180,E1 -25045.354,E2 -25045.354} C_VEL
LIN {X 0,Y 283.076,Z 737.807,A -85,B 0,C 180,E1 -25046.003,E2 -25046.003} C_VEL
LIN {X 0,Y 284.235,Z 704.925,A -85,B 0,C 180,E1 -25047.338,E2 -25047.338} C_VEL
LIN {X 0,Y 285.47,Z 663.236,A -85,B 0,C 180,E1 -25048.972,E2 -25048.972} C_VEL
LIN {X 0,Y 282.883,Z 637.599,A -85,B 0,C 180,E1 -25050.017,E2 -25050.017} C_VEL
LIN {X 0,Y 282.408,Z 629.398,A -85,B 0,C 180,E1 -25050.353,E2 -25050.353} C_VEL
LIN {X 0,Y 282.461,Z 626.49,A -85,B 0,C 180,E1 -25051.382,E2 -25051.382} C_VEL
LIN {X 0,Y 281.7,Z 622.325,A -85,B 0,C 180,E1 -25052.942,E2 -25052.942} C_VEL
LIN {X 0,Y 281.43,Z 622.355,A -85,B 0,C 180,E1 -25057.208,E2 -25057.208} C_VEL
LIN {X 0,Y 281.375,Z 622.368,A -85,B 0,C 180,E1 -25061.685,E2 -25061.685} C_VEL
LIN {X 0,Y 281.409,Z 622.362,A -85,B 0,C 180,E1 -25065.818,E2 -25065.818} C_VEL
LIN {X 0,Y 281.367,Z 622.368,A -85,B 0,C 180,E1 -25069.665,E2 -25069.665} C_VEL
LIN {X 0,Y 281.403,Z 622.362,A -85,B 0,C 180,E1 -25073.317,E2 -25073.317} C_VEL
LIN {X 0,Y 281.393,Z 622.364,A -85,B 0,C 180,E1 -25077.813,E2 -25077.813} C_VEL
LIN {X 0,Y 281.415,Z 622.364,A -85,B 0,C 180,E1 -25081.776,E2 -25081.776} C_VEL
LIN {X 0,Y 281.444,Z 622.354,A -85,B 0,C 180,E1 -25084.97,E2 -25084.97} C_VEL
LIN {X 0,Y 281.448,Z 622.36,A -85,B 0,C 180,E1 -25088.08,E2 -25088.08} C_VEL
LIN {X 0,Y 281.552,Z 622.344,A -85,B 0,C 180,E1 -25091.13,E2 -25091.13} C_VEL
LIN {X 0,Y 281.662,Z 622.33,A -85,B 0,C 180,E1 -25095.895,E2 -25095.895} C_VEL
LIN {X 0,Y 281.679,Z 622.332,A -85,B 0,C 180,E1 -25099.975,E2 -25099.975} C_VEL
LIN {X 0,Y 281.868,Z 622.302,A -85,B 0,C 180,E1 -25104.295,E2 -25104.295} C_VEL
LIN {X 0,Y 281.92,Z 622.296,A -85,B 0,C 180,E1 -25107.151,E2 -25107.151} C_VEL
LIN {X 0,Y 282.041,Z 622.288,A -85,B 0,C 180,E1 -25110,E2 -25110} C_VEL
LIN {X 0,Y 281.942,Z 622.294,A -85,B 0,C 180,E1 -25114.274,E2 -25114.274} C_VEL
LIN {X 0,Y 281.813,Z 622.31,A -85,B 0,C 180,E1 -25117.139,E2 -25117.139} C_VEL
LIN {X 0,Y 281.62,Z 622.336,A -85,B 0,C 180,E1 -25121.477,E2 -25121.477} C_VEL
LIN {X 0,Y 281.619,Z 622.333,A -85,B 0,C 180,E1 -25124.402,E2 -25124.402} C_VEL
LIN {X 0,Y 281.533,Z 622.346,A -85,B 0,C 180,E1 -25129.019,E2 -25129.019} C_VEL
LIN {X 0,Y 281.448,Z 622.355,A -85,B 0,C 180,E1 -25133.465,E2 -25133.465} C_VEL
LIN {X 0,Y 281.423,Z 622.359,A -85,B 0,C 180,E1 -25136.616,E2 -25136.616} C_VEL
LIN {X 0,Y 281.398,Z 622.367,A -85,B 0,C 180,E1 -25139.856,E2 -25139.856} C_VEL
LIN {X 0,Y 281.399,Z 622.36,A -85,B 0,C 180,E1 -25143.203,E2 -25143.203} C_VEL
LIN {X 0,Y 281.462,Z 622.354,A -85,B 0,C 180,E1 -25147.218,E2 -25147.218} C_VEL
LIN {X 0,Y 281.422,Z 622.362,A -85,B 0,C 180,E1 -25151.697,E2 -25151.697} C_VEL
LIN {X 0,Y 281.411,Z 622.362,A -85,B 0,C 180,E1 -25155.82,E2 -25155.82} C_VEL
LIN {X 0,Y 281.409,Z 622.364,A -85,B 0,C 180,E1 -25159.673,E2 -25159.673} C_VEL
LIN {X 0,Y 281.437,Z 622.355,A -85,B 0,C 180,E1 -25163.323,E2 -25163.323} C_VEL
LIN {X 0,Y 281.394,Z 622.366,A -85,B 0,C 180,E1 -25167.814,E2 -25167.814} C_VEL
LIN {X 0,Y 281.416,Z 622.362,A -85,B 0,C 180,E1 -25171.777,E2 -25171.777} C_VEL
LIN {X 0,Y 281.445,Z 622.355,A -85,B 0,C 180,E1 -25174.971,E2 -25174.971} C_VEL
LIN {X 0,Y 281.449,Z 622.361,A -85,B 0,C 180,E1 -25178.081,E2 -25178.081} C_VEL
LIN {X 0,Y 281.504,Z 622.348,A -85,B 0,C 180,E1 -25181.128,E2 -25181.128} C_VEL
LIN {X 0,Y 281.588,Z 622.342,A -85,B 0,C 180,E1 -25185.957,E2 -25185.957} C_VEL
LIN {X 0,Y 281.681,Z 622.331,A -85,B 0,C 180,E1 -25189.976,E2 -25189.976} C_VEL
LIN {X 0,Y 281.952,Z 622.292,A -85,B 0,C 180,E1 -25193.568,E2 -25193.568} C_VEL
LIN {X 0,Y 281.925,Z 622.297,A -85,B 0,C 180,E1 -25197.152,E2 -25197.152} C_VEL
LIN {X 0,Y 282.042,Z 622.286,A -85,B 0,C 180,E1 -25200,E2 -25200} C_VEL
LIN {X 0,Y 281.943,Z 622.297,A -85,B 0,C 180,E1 -25204.275,E2 -25204.275} C_VEL
LIN {X 0,Y 281.817,Z 622.311,A -85,B 0,C 180,E1 -25207.139,E2 -25207.139} C_VEL
LIN {X 0,Y 281.605,Z 622.336,A -85,B 0,C 180,E1 -25211.478,E2 -25211.478} C_VEL
LIN {X 0,Y 281.533,Z 622.347,A -85,B 0,C 180,E1 -25214.407,E2 -25214.407} C_VEL
LIN {X 0,Y 281.449,Z 622.356,A -85,B 0,C 180,E1 -25218.967,E2 -25218.967} C_VEL
LIN {X 0,Y 281.442,Z 622.356,A -85,B 0,C 180,E1 -25223.466,E2 -25223.466} C_VEL
LIN {X 0,Y 281.427,Z 622.36,A -85,B 0,C 180,E1 -25226.616,E2 -25226.616} C_VEL
LIN {X 0,Y 281.391,Z 622.367,A -85,B 0,C 180,E1 -25229.858,E2 -25229.858} C_VEL
LIN {X 0,Y 281.359,Z 622.365,A -85,B 0,C 180,E1 -25233.209,E2 -25233.209} C_VEL
LIN {X 0,Y 281.382,Z 622.365,A -85,B 0,C 180,E1 -25237.196,E2 -25237.196} C_VEL
LIN {X 0,Y 281.357,Z 622.366,A -85,B 0,C 180,E1 -25240.337,E2 -25240.337} C_VEL
LIN {X 0,Y 281.344,Z 622.373,A -85,B 0,C 180,E1 -25244.195,E2 -25244.195} C_VEL
LIN {X 0,Y 281.356,Z 622.369,A -85,B 0,C 180,E1 -25248.319,E2 -25248.319} C_VEL
LIN {X 0,Y 281.353,Z 622.365,A -85,B 0,C 180,E1 -25251.51,E2 -25251.51} C_VEL
LIN {X 0,Y 281.374,Z 622.366,A -85,B 0,C 180,E1 -25255.235,E2 -25255.235} C_VEL
LIN {X 0,Y 281.374,Z 622.365,A -85,B 0,C 180,E1 -25258.482,E2 -25258.482} C_VEL
LIN {X 0,Y 281.477,Z 622.352,A -85,B 0,C 180,E1 -25261.854,E2 -25261.854} C_VEL
LIN {X 0,Y 281.319,Z 622.858,A -85,B 0,C 180,E1 -25262.648,E2 -25262.648} C_VEL
LIN {X 0,Y 280.784,Z 624.15,A -85,B 0,C 180,E1 -25263.403,E2 -25263.403} C_VEL
LIN {X 0,Y 279.043,Z 627.972,A -85,B 0,C 180,E1 -25264.819,E2 -25264.819} C_VEL
LIN {X 0,Y 277.076,Z 632.16,A -85,B 0,C 180,E1 -25266.191,E2 -25266.191} C_VEL
LIN {X 0,Y 275.784,Z 636.349,A -85,B 0,C 180,E1 -25267.594,E2 -25267.594} C_VEL
LIN {X 0,Y 274.915,Z 642.167,A -85,B 0,C 180,E1 -25269.504,E2 -25269.504} C_VEL
LIN {X 0,Y 275.702,Z 661.698,A -85,B 0,C 180,E1 -25270.322,E2 -25270.322} C_VEL
LIN {X 0,Y 277.972,Z 688.632,A -85,B 0,C 180,E1 -25271.45,E2 -25271.45} C_VEL
LIN {X 0,Y 276.182,Z 748.21,A -85,B 0,C 180,E1 -25273.896,E2 -25273.896} C_VEL
LIN {X 0,Y 275.707,Z 759.46,A -85,B 0,C 180,E1 -25274.53,E2 -25274.53} C_VEL
LIN {X 0,Y 275.307,Z 769.357,A -85,B 0,C 180,E1 -25275.261,E2 -25275.261} C_VEL
LIN {X 0,Y 274.902,Z 778.477,A -85,B 0,C 180,E1 -25276.091,E2 -25276.091} C_VEL
LIN {X 0,Y 274.247,Z 789.019,A -85,B 0,C 180,E1 -25277.274,E2 -25277.274} C_VEL
LIN {X 0,Y 273.647,Z 798.454,A -85,B 0,C 180,E1 -25278.558,E2 -25278.558} C_VEL
LIN {X 0,Y 273.101,Z 807.492,A -85,B 0,C 180,E1 -25280.031,E2 -25280.031} C_VEL
LIN {X 0,Y 272.666,Z 815.112,A -85,B 0,C 180,E1 -25281.506,E2 -25281.506} C_VEL
LIN {X 0,Y 272.406,Z 821.668,A -85,B 0,C 180,E1 -25282.985,E2 -25282.985} C_VEL
LIN {X 0,Y 272.202,Z 828.561,A -85,B 0,C 180,E1 -25284.833,E2 -25284.833} C_VEL
LIN {X 0,Y 272.06,Z 833.277,A -85,B 0,C 180,E1 -25286.31,E2 -25286.31} C_VEL
LIN {X 0,Y 271.945,Z 839.043,A -85,B 0,C 180,E1 -25288.524,E2 -25288.524} C_VEL
LIN {X 0,Y 271.837,Z 843.526,A -85,B 0,C 180,E1 -25290.738,E2 -25290.738} C_VEL
LIN {X 0,Y 271.645,Z 846.874,A -85,B 0,C 180,E1 -25292.956,E2 -25292.956} C_VEL
LIN {X 0,Y 271.64,Z 849.701,A -85,B 0,C 180,E1 -25295.92,E2 -25295.92} C_VEL
LIN {X 0,Y 271.895,Z 850.573,A -85,B 0,C 180,E1 -25297.401,E2 -25297.401} C_VEL
LIN {X 0,Y 273.051,Z 851.138,A -85,B 0,C 180,E1 -25300.345,E2 -25300.345} C_VEL
LIN {X 0,Y 275.043,Z 850.037,A -85,B 0,C 180,E1 -25303.25,E2 -25303.25} C_VEL
LIN {X 0,Y 276.35,Z 848.977,A -85,B 0,C 180,E1 -25304.683,E2 -25304.683} C_VEL
LIN {X 0,Y 279.615,Z 845.594,A -85,B 0,C 180,E1 -25307.494,E2 -25307.494} C_VEL
LIN {X 0,Y 282.653,Z 841.913,A -85,B 0,C 180,E1 -25309.545,E2 -25309.545} C_VEL
LIN {X 0,Y 285.97,Z 837.173,A -85,B 0,C 180,E1 -25311.556,E2 -25311.556} C_VEL
LIN {X 0,Y 290.558,Z 830.135,A -85,B 0,C 180,E1 -25313.816,E2 -25313.816} C_VEL
LIN {X 0,Y 294.105,Z 824.075,A -85,B 0,C 180,E1 -25315.385,E2 -25315.385} C_VEL
LIN {X 0,Y 297.945,Z 816.868,A -85,B 0,C 180,E1 -25316.908,E2 -25316.908} C_VEL
LIN {X 0,Y 302.121,Z 808.224,A -85,B 0,C 180,E1 -25318.378,E2 -25318.378} C_VEL
LIN {X 0,Y 306.111,Z 799.112,A -85,B 0,C 180,E1 -25319.659,E2 -25319.659} C_VEL
LIN {X 0,Y 309.764,Z 789.857,A -85,B 0,C 180,E1 -25320.714,E2 -25320.714} C_VEL
LIN {X 0,Y 313.151,Z 780.074,A -85,B 0,C 180,E1 -25321.624,E2 -25321.624} C_VEL
LIN {X 0,Y 316.519,Z 768.679,A -85,B 0,C 180,E1 -25322.463,E2 -25322.463} C_VEL
LIN {X 0,Y 319.264,Z 757.153,A -85,B 0,C 180,E1 -25323.139,E2 -25323.139} C_VEL
LIN {X 0,Y 321.543,Z 745.146,A -85,B 0,C 180,E1 -25323.661,E2 -25323.661} C_VEL
LIN {X 0,Y 326.46,Z 710.944,A -85,B 0,C 180,E1 -25324.923,E2 -25324.923} C_VEL
LIN {X 0,Y 326.273,Z 709.139,A -85,B 0,C 180,E1 -25325.135,E2 -25325.135} C_VEL
LIN {X 0,Y 323.57,Z 701.608,A -85,B 0,C 180,E1 -25326.705,E2 -25326.705} C_VEL
LIN {X 0,Y 320.205,Z 693.634,A -85,B 0,C 180,E1 -25328.908,E2 -25328.908} C_VEL
LIN {X 0,Y 317.727,Z 688.431,A -85,B 0,C 180,E1 -25330.821,E2 -25330.821} C_VEL
LIN {X 0,Y 315.446,Z 683.79,A -85,B 0,C 180,E1 -25333.008,E2 -25333.008} C_VEL
LIN {X 0,Y 312.997,Z 678.909,A -85,B 0,C 180,E1 -25336.649,E2 -25336.649} C_VEL
LIN {X 0,Y 312.592,Z 677.889,A -85,B 0,C 180,E1 -25337.761,E2 -25337.761} C_VEL
LIN {X 0,Y 312.241,Z 677.179,A -85,B 0,C 180,E1 -25339.705,E2 -25339.705} C_VEL
LIN {X 0,Y 312.719,Z 677.314,A -85,B 0,C 180,E1 -25342.788,E2 -25342.788} C_VEL
LIN {X 0,Y 315.239,Z 681.068,A -85,B 0,C 180,E1 -25346.85,E2 -25346.85} C_VEL
LIN {X 0,Y 316.741,Z 683.869,A -85,B 0,C 180,E1 -25348.499,E2 -25348.499} C_VEL
LIN {X 0,Y 318.278,Z 686.104,A -85,B 0,C 180,E1 -25349.705,E2 -25349.705} C_VEL
LIN {X 0,Y 320.725,Z 690.739,A -85,B 0,C 180,E1 -25351.54,E2 -25351.54} C_VEL
LIN {X 0,Y 323.048,Z 695.155,A -85,B 0,C 180,E1 -25352.987,E2 -25352.987} C_VEL
LIN {X 0,Y 325.746,Z 700.948,A -85,B 0,C 180,E1 -25354.529,E2 -25354.529} C_VEL
LIN {X 0,Y 327.084,Z 704.491,A -85,B 0,C 180,E1 -25355.276,E2 -25355.276} C_VEL
LIN {X 0,Y 321.599,Z 740.898,A -85,B 0,C 180,E1 -25356.592,E2 -25356.592} C_VEL
LIN {X 0,Y 318.763,Z 755.379,A -85,B 0,C 180,E1 -25357.316,E2 -25357.316} C_VEL
LIN {X 0,Y 315.555,Z 767.723,A -85,B 0,C 180,E1 -25358.173,E2 -25358.173} C_VEL
LIN {X 0,Y 312.233,Z 778.427,A -85,B 0,C 180,E1 -25359.137,E2 -25359.137} C_VEL
LIN {X 0,Y 308.545,Z 788.531,A -85,B 0,C 180,E1 -25360.264,E2 -25360.264} C_VEL
LIN {X 0,Y 305.491,Z 796.042,A -85,B 0,C 180,E1 -25361.276,E2 -25361.276} C_VEL
LIN {X 0,Y 301.199,Z 805.386,A -85,B 0,C 180,E1 -25362.808,E2 -25362.808} C_VEL
LIN {X 0,Y 297.436,Z 812.773,A -85,B 0,C 180,E1 -25364.287,E2 -25364.287} C_VEL
LIN {X 0,Y 293.72,Z 819.229,A -85,B 0,C 180,E1 -25365.851,E2 -25365.851} C_VEL
LIN {X 0,Y 290.256,Z 824.648,A -85,B 0,C 180,E1 -25367.456,E2 -25367.456} C_VEL
LIN {X 0,Y 286.456,Z 829.926,A -85,B 0,C 180,E1 -25369.432,E2 -25369.432} C_VEL
LIN {X 0,Y 283.062,Z 834.109,A -85,B 0,C 180,E1 -25371.461,E2 -25371.461} C_VEL
LIN {X 0,Y 281.044,Z 836.367,A -85,B 0,C 180,E1 -25372.841,E2 -25372.841} C_VEL
LIN {X 0,Y 277.533,Z 839.371,A -85,B 0,C 180,E1 -25375.657,E2 -25375.657} C_VEL
LIN {X 0,Y 276.096,Z 840.26,A -85,B 0,C 180,E1 -25377.091,E2 -25377.091} C_VEL
LIN {X 0,Y 273.912,Z 840.898,A -85,B 0,C 180,E1 -25380,E2 -25380} C_VEL
LIN {X 0,Y 272.402,Z 839.804,A -85,B 0,C 180,E1 -25382.947,E2 -25382.947} C_VEL
LIN {X 0,Y 271.897,Z 838.728,A -85,B 0,C 180,E1 -25384.432,E2 -25384.432} C_VEL
LIN {X 0,Y 271.253,Z 835.218,A -85,B 0,C 180,E1 -25387.418,E2 -25387.418} C_VEL
LIN {X 0,Y 271.264,Z 831.39,A -85,B 0,C 180,E1 -25389.662,E2 -25389.662} C_VEL
LIN {X 0,Y 271.361,Z 826.348,A -85,B 0,C 180,E1 -25391.917,E2 -25391.917} C_VEL
LIN {X 0,Y 271.657,Z 819.95,A -85,B 0,C 180,E1 -25394.178,E2 -25394.178} C_VEL
LIN {X 0,Y 272.015,Z 813.426,A -85,B 0,C 180,E1 -25396.07,E2 -25396.07} C_VEL
LIN {X 0,Y 272.382,Z 805.481,A -85,B 0,C 180,E1 -25397.973,E2 -25397.973} C_VEL
LIN {X 0,Y 272.826,Z 797.969,A -85,B 0,C 180,E1 -25399.496,E2 -25399.496} C_VEL
LIN {X 0,Y 273.334,Z 789.033,A -85,B 0,C 180,E1 -25401.024,E2 -25401.024} C_VEL
LIN {X 0,Y 273.896,Z 779.679,A -85,B 0,C 180,E1 -25402.358,E2 -25402.358} C_VEL
LIN {X 0,Y 274.543,Z 769.984,A -85,B 0,C 180,E1 -25403.508,E2 -25403.508} C_VEL
LIN {X 0,Y 275.084,Z 759.302,A -85,B 0,C 180,E1 -25404.542,E2 -25404.542} C_VEL
LIN {X 0,Y 275.574,Z 749.613,A -85,B 0,C 180,E1 -25405.298,E2 -25405.298} C_VEL
LIN {X 0,Y 275.942,Z 738.471,A -85,B 0,C 180,E1 -25405.967,E2 -25405.967} C_VEL
LIN {X 0,Y 276.884,Z 712.06,A -85,B 0,C 180,E1 -25407.087,E2 -25407.087} C_VEL
LIN {X 0,Y 278.358,Z 663.556,A -85,B 0,C 180,E1 -25409.044,E2 -25409.044} C_VEL
LIN {X 0,Y 275.839,Z 638.124,A -85,B 0,C 180,E1 -25410.121,E2 -25410.121} C_VEL
LIN {X 0,Y 275.354,Z 629.452,A -85,B 0,C 180,E1 -25410.514,E2 -25410.514} C_VEL
LIN {X 0,Y 275.357,Z 626.927,A -85,B 0,C 180,E1 -25411.43,E2 -25411.43} C_VEL
LIN {X 0,Y 274.662,Z 623.202,A -85,B 0,C 180,E1 -25412.835,E2 -25412.835} C_VEL
LIN {X 0,Y 274.363,Z 623.239,A -85,B 0,C 180,E1 -25417.785,E2 -25417.785} C_VEL
LIN {X 0,Y 274.326,Z 623.246,A -85,B 0,C 180,E1 -25422.228,E2 -25422.228} C_VEL
LIN {X 0,Y 274.37,Z 623.238,A -85,B 0,C 180,E1 -25425.627,E2 -25425.627} C_VEL
LIN {X 0,Y 274.331,Z 623.247,A -85,B 0,C 180,E1 -25429.993,E2 -25429.993} C_VEL
LIN {X 0,Y 274.339,Z 623.244,A -85,B 0,C 180,E1 -25434.038,E2 -25434.038} C_VEL
LIN {X 0,Y 274.342,Z 623.241,A -85,B 0,C 180,E1 -25437.576,E2 -25437.576} C_VEL
LIN {X 0,Y 274.343,Z 623.242,A -85,B 0,C 180,E1 -25440.98,E2 -25440.98} C_VEL
LIN {X 0,Y 274.375,Z 623.237,A -85,B 0,C 180,E1 -25444.279,E2 -25444.279} C_VEL
LIN {X 0,Y 274.407,Z 623.232,A -85,B 0,C 180,E1 -25447.487,E2 -25447.487} C_VEL
LIN {X 0,Y 274.472,Z 623.226,A -85,B 0,C 180,E1 -25450.772,E2 -25450.772} C_VEL
LIN {X 0,Y 274.619,Z 623.206,A -85,B 0,C 180,E1 -25455.746,E2 -25455.746} C_VEL
LIN {X 0,Y 274.618,Z 623.21,A -85,B 0,C 180,E1 -25459.715,E2 -25459.715} C_VEL
LIN {X 0,Y 274.837,Z 623.179,A -85,B 0,C 180,E1 -25464.149,E2 -25464.149} C_VEL
LIN {X 0,Y 274.958,Z 623.166,A -85,B 0,C 180,E1 -25468.54,E2 -25468.54} C_VEL
LIN {X 0,Y 274.957,Z 623.166,A -85,B 0,C 180,E1 -25471.459,E2 -25471.459} C_VEL
LIN {X 0,Y 274.837,Z 623.179,A -85,B 0,C 180,E1 -25475.851,E2 -25475.851} C_VEL
LIN {X 0,Y 274.617,Z 623.21,A -85,B 0,C 180,E1 -25480.285,E2 -25480.285} C_VEL
LIN {X 0,Y 274.618,Z 623.206,A -85,B 0,C 180,E1 -25484.253,E2 -25484.253} C_VEL
LIN {X 0,Y 274.464,Z 623.227,A -85,B 0,C 180,E1 -25489.376,E2 -25489.376} C_VEL
LIN {X 0,Y 274.416,Z 623.23,A -85,B 0,C 180,E1 -25493.237,E2 -25493.237} C_VEL
LIN {X 0,Y 274.357,Z 623.24,A -85,B 0,C 180,E1 -25497.358,E2 -25497.358} C_VEL
LIN {X 0,Y 274.333,Z 623.243,A -85,B 0,C 180,E1 -25500.707,E2 -25500.707} C_VEL
LIN {X 0,Y 274.379,Z 623.237,A -85,B 0,C 180,E1 -25504.168,E2 -25504.168} C_VEL
LIN {X 0,Y 274.412,Z 623.235,A -85,B 0,C 180,E1 -25507.778,E2 -25507.778} C_VEL
LIN {X 0,Y 274.388,Z 623.237,A -85,B 0,C 180,E1 -25511.583,E2 -25511.583} C_VEL
LIN {X 0,Y 274.371,Z 623.237,A -85,B 0,C 180,E1 -25515.628,E2 -25515.628} C_VEL
LIN {X 0,Y 274.378,Z 623.242,A -85,B 0,C 180,E1 -25519.983,E2 -25519.983} C_VEL
LIN {X 0,Y 274.411,Z 623.232,A -85,B 0,C 180,E1 -25522.306,E2 -25522.306} C_VEL
LIN {X 0,Y 274.339,Z 623.243,A -85,B 0,C 180,E1 -25525.827,E2 -25525.827} C_VEL
LIN {X 0,Y 274.349,Z 623.243,A -85,B 0,C 180,E1 -25530.233,E2 -25530.233} C_VEL
LIN {X 0,Y 274.376,Z 623.238,A -85,B 0,C 180,E1 -25534.28,E2 -25534.28} C_VEL
LIN {X 0,Y 274.408,Z 623.234,A -85,B 0,C 180,E1 -25537.488,E2 -25537.488} C_VEL
LIN {X 0,Y 274.461,Z 623.225,A -85,B 0,C 180,E1 -25540.78,E2 -25540.78} C_VEL
LIN {X 0,Y 274.544,Z 623.218,A -85,B 0,C 180,E1 -25545.811,E2 -25545.811} C_VEL
LIN {X 0,Y 274.617,Z 623.21,A -85,B 0,C 180,E1 -25549.716,E2 -25549.716} C_VEL
LIN {X 0,Y 274.861,Z 623.18,A -85,B 0,C 180,E1 -25554.15,E2 -25554.15} C_VEL
LIN {X 0,Y 274.961,Z 623.165,A -85,B 0,C 180,E1 -25558.541,E2 -25558.541} C_VEL
LIN {X 0,Y 274.945,Z 623.165,A -85,B 0,C 180,E1 -25561.46,E2 -25561.46} C_VEL
LIN {X 0,Y 274.899,Z 623.173,A -85,B 0,C 180,E1 -25564.384,E2 -25564.384} C_VEL
LIN {X 0,Y 274.756,Z 623.191,A -85,B 0,C 180,E1 -25567.324,E2 -25567.324} C_VEL
LIN {X 0,Y 274.545,Z 623.217,A -85,B 0,C 180,E1 -25571.777,E2 -25571.777} C_VEL
LIN {X 0,Y 274.465,Z 623.226,A -85,B 0,C 180,E1 -25574.786,E2 -25574.786} C_VEL
LIN {X 0,Y 274.393,Z 623.235,A -85,B 0,C 180,E1 -25579.382,E2 -25579.382} C_VEL
LIN {X 0,Y 274.408,Z 623.231,A -85,B 0,C 180,E1 -25583.231,E2 -25583.231} C_VEL
LIN {X 0,Y 274.36,Z 623.24,A -85,B 0,C 180,E1 -25587.358,E2 -25587.358} C_VEL
LIN {X 0,Y 274.31,Z 623.242,A -85,B 0,C 180,E1 -25590.71,E2 -25590.71} C_VEL
LIN {X 0,Y 274.327,Z 623.247,A -85,B 0,C 180,E1 -25594.176,E2 -25594.176} C_VEL
LIN {X 0,Y 274.316,Z 623.248,A -85,B 0,C 180,E1 -25597.794,E2 -25597.794} C_VEL
LIN {X 0,Y 274.33,Z 623.241,A -85,B 0,C 180,E1 -25601.595,E2 -25601.595} C_VEL
LIN {X 0,Y 274.289,Z 623.25,A -85,B 0,C 180,E1 -25605.646,E2 -25605.646} C_VEL
LIN {X 0,Y 274.33,Z 623.244,A -85,B 0,C 180,E1 -25608.406,E2 -25608.406} C_VEL
LIN {X 0,Y 274.318,Z 623.245,A -85,B 0,C 180,E1 -25612.331,E2 -25612.331} C_VEL
LIN {X 0,Y 274.325,Z 623.247,A -85,B 0,C 180,E1 -25615.824,E2 -25615.824} C_VEL
LIN {X 0,Y 274.345,Z 623.24,A -85,B 0,C 180,E1 -25620.236,E2 -25620.236} C_VEL
LIN {X 0,Y 274.591,Z 623.399,A -85,B 0,C 180,E1 -25623.097,E2 -25623.097} C_VEL
LIN {X 0,Y 276.13,Z 631.833,A -85,B 0,C 180,E1 -25626.055,E2 -25626.055} C_VEL
LIN {X 0,Y 275.951,Z 635.266,A -85,B 0,C 180,E1 -25627.227,E2 -25627.227} C_VEL
LIN {X 0,Y 275.784,Z 636.349,A -85,B 0,C 180,E1 -25627.594,E2 -25627.594} C_VEL
LIN {X 0,Y 275.208,Z 638.703,A -85,B 0,C 180,E1 -25628.218,E2 -25628.218} C_VEL
LIN {X 0,Y 273.645,Z 643.117,A -85,B 0,C 180,E1 -25628.946,E2 -25628.946} C_VEL
LIN {X 0,Y 271.756,Z 648.145,A -85,B 0,C 180,E1 -25629.465,E2 -25629.465} C_VEL
LIN {X 0,Y 269.484,Z 655.617,A -85,B 0,C 180,E1 -25629.948,E2 -25629.948} C_VEL
LIN {X 0,Y 268.699,Z 661.491,A -85,B 0,C 180,E1 -25630.223,E2 -25630.223} C_VEL
LIN {X 0,Y 268.731,Z 663.472,A -85,B 0,C 180,E1 -25630.309,E2 -25630.309} C_VEL
LIN {X 0,Y 270.861,Z 689.675,A -85,B 0,C 180,E1 -25631.434,E2 -25631.434} C_VEL
LIN {X 0,Y 269.111,Z 747.822,A -85,B 0,C 180,E1 -25633.897,E2 -25633.897} C_VEL
LIN {X 0,Y 268.625,Z 758.949,A -85,B 0,C 180,E1 -25634.537,E2 -25634.537} C_VEL
LIN {X 0,Y 268.203,Z 769.6,A -85,B 0,C 180,E1 -25635.348,E2 -25635.348} C_VEL
LIN {X 0,Y 267.794,Z 778.921,A -85,B 0,C 180,E1 -25636.237,E2 -25636.237} C_VEL
LIN {X 0,Y 267.198,Z 788.253,A -85,B 0,C 180,E1 -25637.318,E2 -25637.318} C_VEL
LIN {X 0,Y 266.616,Z 797.715,A -85,B 0,C 180,E1 -25638.637,E2 -25638.637} C_VEL
LIN {X 0,Y 266.079,Z 806.771,A -85,B 0,C 180,E1 -25640.148,E2 -25640.148} C_VEL
LIN {X 0,Y 265.628,Z 814.442,A -85,B 0,C 180,E1 -25641.661,E2 -25641.661} C_VEL
LIN {X 0,Y 265.388,Z 821.08,A -85,B 0,C 180,E1 -25643.179,E2 -25643.179} C_VEL
LIN {X 0,Y 265.183,Z 828.037,A -85,B 0,C 180,E1 -25645.076,E2 -25645.076} C_VEL
LIN {X 0,Y 265.061,Z 833.837,A -85,B 0,C 180,E1 -25646.971,E2 -25646.971} C_VEL
LIN {X 0,Y 264.926,Z 839.403,A -85,B 0,C 180,E1 -25649.243,E2 -25649.243} C_VEL
LIN {X 0,Y 264.78,Z 843.726,A -85,B 0,C 180,E1 -25651.516,E2 -25651.516} C_VEL
LIN {X 0,Y 264.617,Z 845.929,A -85,B 0,C 180,E1 -25653.035,E2 -25653.035} C_VEL
LIN {X 0,Y 264.6,Z 849.153,A -85,B 0,C 180,E1 -25656.079,E2 -25656.079} C_VEL
LIN {X 0,Y 265.341,Z 850.676,A -85,B 0,C 180,E1 -25659.114,E2 -25659.114} C_VEL
LIN {X 0,Y 266.073,Z 850.906,A -85,B 0,C 180,E1 -25660.619,E2 -25660.619} C_VEL
LIN {X 0,Y 268.136,Z 850.216,A -85,B 0,C 180,E1 -25663.598,E2 -25663.598} C_VEL
LIN {X 0,Y 271.145,Z 847.867,A -85,B 0,C 180,E1 -25666.509,E2 -25666.509} C_VEL
LIN {X 0,Y 273.928,Z 845.102,A -85,B 0,C 180,E1 -25668.641,E2 -25668.641} C_VEL
LIN {X 0,Y 277.097,Z 841.39,A -85,B 0,C 180,E1 -25670.726,E2 -25670.726} C_VEL
LIN {X 0,Y 280.789,Z 836.633,A -85,B 0,C 180,E1 -25672.747,E2 -25672.747} C_VEL
LIN {X 0,Y 284.919,Z 830.672,A -85,B 0,C 180,E1 -25674.704,E2 -25674.704} C_VEL
LIN {X 0,Y 289.414,Z 823.329,A -85,B 0,C 180,E1 -25676.599,E2 -25676.599} C_VEL
LIN {X 0,Y 293.498,Z 816.104,A -85,B 0,C 180,E1 -25678.122,E2 -25678.122} C_VEL
LIN {X 0,Y 297.891,Z 807.507,A -85,B 0,C 180,E1 -25679.59,E2 -25679.59} C_VEL
LIN {X 0,Y 302.07,Z 798.294,A -85,B 0,C 180,E1 -25680.867,E2 -25680.867} C_VEL
LIN {X 0,Y 305.97,Z 788.75,A -85,B 0,C 180,E1 -25681.921,E2 -25681.921} C_VEL
LIN {X 0,Y 309.295,Z 779.405,A -85,B 0,C 180,E1 -25682.771,E2 -25682.771} C_VEL
LIN {X 0,Y 312.429,Z 769.482,A -85,B 0,C 180,E1 -25683.51,E2 -25683.51} C_VEL
LIN {X 0,Y 315.57,Z 757.223,A -85,B 0,C 180,E1 -25684.239,E2 -25684.239} C_VEL
LIN {X 0,Y 317.928,Z 745.635,A -85,B 0,C 180,E1 -25684.751,E2 -25684.751} C_VEL
LIN {X 0,Y 322.767,Z 713.502,A -85,B 0,C 180,E1 -25685.932,E2 -25685.932} C_VEL
LIN {X 0,Y 320.591,Z 706.98,A -85,B 0,C 180,E1 -25687.354,E2 -25687.354} C_VEL
LIN {X 0,Y 317.58,Z 699.479,A -85,B 0,C 180,E1 -25689.471,E2 -25689.471} C_VEL
LIN {X 0,Y 315.382,Z 694.61,A -85,B 0,C 180,E1 -25691.306,E2 -25691.306} C_VEL
LIN {X 0,Y 313.377,Z 690.237,A -85,B 0,C 180,E1 -25693.425,E2 -25693.425} C_VEL
LIN {X 0,Y 311.031,Z 684.959,A -85,B 0,C 180,E1 -25697.499,E2 -25697.499} C_VEL
LIN {X 0,Y 310.574,Z 684.05,A -85,B 0,C 180,E1 -25700.069,E2 -25700.069} C_VEL
LIN {X 0,Y 311.071,Z 684.226,A -85,B 0,C 180,E1 -25702.711,E2 -25702.711} C_VEL
LIN {X 0,Y 313.416,Z 687.884,A -85,B 0,C 180,E1 -25706.688,E2 -25706.688} C_VEL
LIN {X 0,Y 316.088,Z 692.617,A -85,B 0,C 180,E1 -25709.358,E2 -25709.358} C_VEL
LIN {X 0,Y 318.304,Z 697.032,A -85,B 0,C 180,E1 -25711.142,E2 -25711.142} C_VEL
LIN {X 0,Y 321.137,Z 702.688,A -85,B 0,C 180,E1 -25712.973,E2 -25712.973} C_VEL
LIN {X 0,Y 323.258,Z 707.821,A -85,B 0,C 180,E1 -25714.273,E2 -25714.273} C_VEL
LIN {X 0,Y 317.983,Z 741.76,A -85,B 0,C 180,E1 -25715.511,E2 -25715.511} C_VEL
LIN {X 0,Y 315.083,Z 755.678,A -85,B 0,C 180,E1 -25716.217,E2 -25716.217} C_VEL
LIN {X 0,Y 311.361,Z 768.898,A -85,B 0,C 180,E1 -25717.148,E2 -25717.148} C_VEL
LIN {X 0,Y 307.854,Z 779.483,A -85,B 0,C 180,E1 -25718.125,E2 -25718.125} C_VEL
LIN {X 0,Y 304.482,Z 788.37,A -85,B 0,C 180,E1 -25719.11,E2 -25719.11} C_VEL
LIN {X 0,Y 300.837,Z 796.922,A -85,B 0,C 180,E1 -25720.269,E2 -25720.269} C_VEL
LIN {X 0,Y 297.322,Z 804.273,A -85,B 0,C 180,E1 -25721.455,E2 -25721.455} C_VEL
LIN {X 0,Y 292.827,Z 812.55,A -85,B 0,C 180,E1 -25723.099,E2 -25723.099} C_VEL
LIN {X 0,Y 288.476,Z 819.744,A -85,B 0,C 180,E1 -25724.869,E2 -25724.869} C_VEL
LIN {X 0,Y 284.807,Z 825.135,A -85,B 0,C 180,E1 -25726.488,E2 -25726.488} C_VEL
LIN {X 0,Y 282.079,Z 828.853,A -85,B 0,C 180,E1 -25727.815,E2 -25727.815} C_VEL
LIN {X 0,Y 278.351,Z 833.296,A -85,B 0,C 180,E1 -25729.854,E2 -25729.854} C_VEL
LIN {X 0,Y 273.976,Z 837.528,A -85,B 0,C 180,E1 -25732.655,E2 -25732.655} C_VEL
LIN {X 0,Y 272.118,Z 839.091,A -85,B 0,C 180,E1 -25734.09,E2 -25734.09} C_VEL
LIN {X 0,Y 268.989,Z 840.817,A -85,B 0,C 180,E1 -25737.014,E2 -25737.014} C_VEL
LIN {X 0,Y 266.756,Z 840.9,A -85,B 0,C 180,E1 -25740,E2 -25740} C_VEL
LIN {X 0,Y 265.935,Z 840.463,A -85,B 0,C 180,E1 -25741.509,E2 -25741.509} C_VEL
LIN {X 0,Y 264.756,Z 838.137,A -85,B 0,C 180,E1 -25744.552,E2 -25744.552} C_VEL
LIN {X 0,Y 264.247,Z 835.342,A -85,B 0,C 180,E1 -25746.85,E2 -25746.85} C_VEL
LIN {X 0,Y 264.199,Z 831.547,A -85,B 0,C 180,E1 -25749.152,E2 -25749.152} C_VEL
LIN {X 0,Y 264.315,Z 826.932,A -85,B 0,C 180,E1 -25751.327,E2 -25751.327} C_VEL
LIN {X 0,Y 264.539,Z 820.178,A -85,B 0,C 180,E1 -25753.786,E2 -25753.786} C_VEL
LIN {X 0,Y 264.914,Z 813.681,A -85,B 0,C 180,E1 -25755.724,E2 -25755.724} C_VEL
LIN {X 0,Y 265.237,Z 806.54,A -85,B 0,C 180,E1 -25757.505,E2 -25757.505} C_VEL
LIN {X 0,Y 265.738,Z 798.284,A -85,B 0,C 180,E1 -25759.237,E2 -25759.237} C_VEL
LIN {X 0,Y 266.234,Z 789.377,A -85,B 0,C 180,E1 -25760.804,E2 -25760.804} C_VEL
LIN {X 0,Y 266.785,Z 780.113,A -85,B 0,C 180,E1 -25762.173,E2 -25762.173} C_VEL
LIN {X 0,Y 267.475,Z 769.539,A -85,B 0,C 180,E1 -25763.466,E2 -25763.466} C_VEL
LIN {X 0,Y 267.977,Z 760.058,A -85,B 0,C 180,E1 -25764.42,E2 -25764.42} C_VEL
LIN {X 0,Y 268.492,Z 749.322,A -85,B 0,C 180,E1 -25765.289,E2 -25765.289} C_VEL
LIN {X 0,Y 268.848,Z 738.187,A -85,B 0,C 180,E1 -25765.977,E2 -25765.977} C_VEL
LIN {X 0,Y 269.978,Z 707.326,A -85,B 0,C 180,E1 -25767.315,E2 -25767.315} C_VEL
LIN {X 0,Y 271.269,Z 663.999,A -85,B 0,C 180,E1 -25769.114,E2 -25769.114} C_VEL
LIN {X 0,Y 268.534,Z 635.692,A -85,B 0,C 180,E1 -25770.346,E2 -25770.346} C_VEL
LIN {X 0,Y 268.291,Z 629.697,A -85,B 0,C 180,E1 -25770.622,E2 -25770.622} C_VEL
LIN {X 0,Y 268.068,Z 626.312,A -85,B 0,C 180,E1 -25771.886,E2 -25771.886} C_VEL
LIN {X 0,Y 267.63,Z 624.078,A -85,B 0,C 180,E1 -25772.777,E2 -25772.777} C_VEL
LIN {X 0,Y 267.3,Z 624.115,A -85,B 0,C 180,E1 -25777.063,E2 -25777.063} C_VEL
LIN {X 0,Y 267.289,Z 624.12,A -85,B 0,C 180,E1 -25780.929,E2 -25780.929} C_VEL
LIN {X 0,Y 267.324,Z 624.113,A -85,B 0,C 180,E1 -25785.027,E2 -25785.027} C_VEL
LIN {X 0,Y 267.287,Z 624.121,A -85,B 0,C 180,E1 -25789.46,E2 -25789.46} C_VEL
LIN {X 0,Y 267.307,Z 624.117,A -85,B 0,C 180,E1 -25794.322,E2 -25794.322} C_VEL
LIN {X 0,Y 267.274,Z 624.123,A -85,B 0,C 180,E1 -25798.389,E2 -25798.389} C_VEL
LIN {X 0,Y 267.304,Z 624.122,A -85,B 0,C 180,E1 -25801.857,E2 -25801.857} C_VEL
LIN {X 0,Y 267.305,Z 624.115,A -85,B 0,C 180,E1 -25805.212,E2 -25805.212} C_VEL
LIN {X 0,Y 267.342,Z 624.115,A -85,B 0,C 180,E1 -25808.481,E2 -25808.481} C_VEL
LIN {X 0,Y 267.416,Z 624.107,A -85,B 0,C 180,E1 -25811.68,E2 -25811.68} C_VEL
LIN {X 0,Y 267.572,Z 624.085,A -85,B 0,C 180,E1 -25816.373,E2 -25816.373} C_VEL
LIN {X 0,Y 267.628,Z 624.078,A -85,B 0,C 180,E1 -25820.965,E2 -25820.965} C_VEL
LIN {X 0,Y 267.811,Z 624.056,A -85,B 0,C 180,E1 -25823.995,E2 -25823.995} C_VEL
LIN {X 0,Y 267.907,Z 624.044,A -85,B 0,C 180,E1 -25828.502,E2 -25828.502} C_VEL
LIN {X 0,Y 267.907,Z 624.044,A -85,B 0,C 180,E1 -25831.498,E2 -25831.498} C_VEL
LIN {X 0,Y 267.811,Z 624.056,A -85,B 0,C 180,E1 -25836.005,E2 -25836.005} C_VEL
LIN {X 0,Y 267.549,Z 624.089,A -85,B 0,C 180,E1 -25840.559,E2 -25840.559} C_VEL
LIN {X 0,Y 267.55,Z 624.086,A -85,B 0,C 180,E1 -25844.386,E2 -25844.386} C_VEL
LIN {X 0,Y 267.425,Z 624.104,A -85,B 0,C 180,E1 -25849.455,E2 -25849.455} C_VEL
LIN {X 0,Y 267.352,Z 624.111,A -85,B 0,C 180,E1 -25853.514,E2 -25853.514} C_VEL
LIN {X 0,Y 267.319,Z 624.116,A -85,B 0,C 180,E1 -25857.017,E2 -25857.017} C_VEL
LIN {X 0,Y 267.292,Z 624.123,A -85,B 0,C 180,E1 -25860.145,E2 -25860.145} C_VEL
LIN {X 0,Y 267.319,Z 624.114,A -85,B 0,C 180,E1 -25863.384,E2 -25863.384} C_VEL
LIN {X 0,Y 267.35,Z 624.112,A -85,B 0,C 180,E1 -25867.055,E2 -25867.055} C_VEL
LIN {X 0,Y 267.323,Z 624.115,A -85,B 0,C 180,E1 -25870.924,E2 -25870.924} C_VEL
LIN {X 0,Y 267.323,Z 624.113,A -85,B 0,C 180,E1 -25875.028,E2 -25875.028} C_VEL
LIN {X 0,Y 267.321,Z 624.117,A -85,B 0,C 180,E1 -25879.452,E2 -25879.452} C_VEL
LIN {X 0,Y 267.319,Z 624.113,A -85,B 0,C 180,E1 -25882.94,E2 -25882.94} C_VEL
LIN {X 0,Y 267.305,Z 624.118,A -85,B 0,C 180,E1 -25886.985,E2 -25886.985} C_VEL
LIN {X 0,Y 267.303,Z 624.121,A -85,B 0,C 180,E1 -25890.141,E2 -25890.141} C_VEL
LIN {X 0,Y 267.357,Z 624.109,A -85,B 0,C 180,E1 -25893.553,E2 -25893.553} C_VEL
LIN {X 0,Y 267.392,Z 624.107,A -85,B 0,C 180,E1 -25896.864,E2 -25896.864} C_VEL
LIN {X 0,Y 267.396,Z 624.108,A -85,B 0,C 180,E1 -25901.68,E2 -25901.68} C_VEL
LIN {X 0,Y 267.514,Z 624.094,A -85,B 0,C 180,E1 -25906.371,E2 -25906.371} C_VEL
LIN {X 0,Y 267.633,Z 624.075,A -85,B 0,C 180,E1 -25910.966,E2 -25910.966} C_VEL
LIN {X 0,Y 267.824,Z 624.054,A -85,B 0,C 180,E1 -25913.996,E2 -25913.996} C_VEL
LIN {X 0,Y 267.86,Z 624.049,A -85,B 0,C 180,E1 -25917.003,E2 -25917.003} C_VEL
LIN {X 0,Y 268.002,Z 624.034,A -85,B 0,C 180,E1 -25920,E2 -25920} C_VEL
LIN {X 0,Y 267.858,Z 624.05,A -85,B 0,C 180,E1 -25924.5,E2 -25924.5} C_VEL
LIN {X 0,Y 267.702,Z 624.07,A -85,B 0,C 180,E1 -25927.518,E2 -25927.518} C_VEL
LIN {X 0,Y 267.488,Z 624.095,A -85,B 0,C 180,E1 -25932.093,E2 -25932.093} C_VEL
LIN {X 0,Y 267.403,Z 624.105,A -85,B 0,C 180,E1 -25935.186,E2 -25935.186} C_VEL
LIN {X 0,Y 267.345,Z 624.113,A -85,B 0,C 180,E1 -25939.405,E2 -25939.405} C_VEL
LIN {X 0,Y 267.345,Z 624.112,A -85,B 0,C 180,E1 -25943.509,E2 -25943.509} C_VEL
LIN {X 0,Y 267.323,Z 624.116,A -85,B 0,C 180,E1 -25947.017,E2 -25947.017} C_VEL
LIN {X 0,Y 267.278,Z 624.122,A -85,B 0,C 180,E1 -25950.138,E2 -25950.138} C_VEL
LIN {X 0,Y 267.289,Z 624.119,A -85,B 0,C 180,E1 -25953.389,E2 -25953.389} C_VEL
LIN {X 0,Y 267.254,Z 624.125,A -85,B 0,C 180,E1 -25957.071,E2 -25957.071} C_VEL
LIN {X 0,Y 267.279,Z 624.117,A -85,B 0,C 180,E1 -25960.932,E2 -25960.932} C_VEL
LIN {X 0,Y 267.23,Z 624.127,A -85,B 0,C 180,E1 -25965.049,E2 -25965.049} C_VEL
LIN {X 0,Y 267.279,Z 624.12,A -85,B 0,C 180,E1 -25969.068,E2 -25969.068} C_VEL
LIN {X 0,Y 267.253,Z 624.123,A -85,B 0,C 180,E1 -25972.929,E2 -25972.929} C_VEL
LIN {X 0,Y 267.296,Z 624.119,A -85,B 0,C 180,E1 -25976.988,E2 -25976.988} C_VEL
LIN {X 0,Y 267.392,Z 624.107,A -85,B 0,C 180,E1 -25981.867,E2 -25981.867} C_VEL
LIN {X 0,Y 267.545,Z 624.26,A -85,B 0,C 180,E1 -25983.152,E2 -25983.152} C_VEL
LIN {X 0,Y 268.924,Z 631.421,A -85,B 0,C 180,E1 -25985.73,E2 -25985.73} C_VEL
LIN {X 0,Y 269.125,Z 633.274,A -85,B 0,C 180,E1 -25986.387,E2 -25986.387} C_VEL
LIN {X 0,Y 267.849,Z 641.875,A -85,B 0,C 180,E1 -25989.38,E2 -25989.38} C_VEL
LIN {X 0,Y 268.512,Z 660.417,A -85,B 0,C 180,E1 -25990.177,E2 -25990.177} C_VEL
LIN {X 0,Y 268.731,Z 663.472,A -85,B 0,C 180,E1 -25990.309,E2 -25990.309} C_VEL
LIN {X 0,Y 268.537,Z 669.268,A -85,B 0,C 180,E1 -25990.552,E2 -25990.552} C_VEL
LIN {X 0,Y 264.041,Z 690.28,A -85,B 0,C 180,E1 -25991.402,E2 -25991.402} C_VEL
LIN {X 0,Y 263.639,Z 694.162,A -85,B 0,C 180,E1 -25991.567,E2 -25991.567} C_VEL
LIN {X 0,Y 262.056,Z 746.923,A -85,B 0,C 180,E1 -25993.9,E2 -25993.9} C_VEL
LIN {X 0,Y 261.549,Z 758.719,A -85,B 0,C 180,E1 -25994.602,E2 -25994.602} C_VEL
LIN {X 0,Y 261.157,Z 768.838,A -85,B 0,C 180,E1 -25995.394,E2 -25995.394} C_VEL
LIN {X 0,Y 260.7,Z 779.107,A -85,B 0,C 180,E1 -25996.403,E2 -25996.403} C_VEL
LIN {X 0,Y 260.089,Z 788.7,A -85,B 0,C 180,E1 -25997.559,E2 -25997.559} C_VEL
LIN {X 0,Y 259.555,Z 798.073,A -85,B 0,C 180,E1 -25998.915,E2 -25998.915} C_VEL
LIN {X 0,Y 258.997,Z 807.026,A -85,B 0,C 180,E1 -26000.465,E2 -26000.465} C_VEL
LIN {X 0,Y 258.592,Z 813.771,A -85,B 0,C 180,E1 -26001.825,E2 -26001.825} C_VEL
LIN {X 0,Y 258.341,Z 821.926,A -85,B 0,C 180,E1 -26003.774,E2 -26003.774} C_VEL
LIN {X 0,Y 258.144,Z 828.699,A -85,B 0,C 180,E1 -26005.721,E2 -26005.721} C_VEL
LIN {X 0,Y 258.061,Z 834.333,A -85,B 0,C 180,E1 -26007.667,E2 -26007.667} C_VEL
LIN {X 0,Y 257.942,Z 838.102,A -85,B 0,C 180,E1 -26009.222,E2 -26009.222} C_VEL
LIN {X 0,Y 257.769,Z 842.63,A -85,B 0,C 180,E1 -26011.557,E2 -26011.557} C_VEL
LIN {X 0,Y 257.535,Z 846.914,A -85,B 0,C 180,E1 -26014.681,E2 -26014.681} C_VEL
LIN {X 0,Y 257.567,Z 848.428,A -85,B 0,C 180,E1 -26016.245,E2 -26016.245} C_VEL
LIN {X 0,Y 258.344,Z 850.346,A -85,B 0,C 180,E1 -26019.363,E2 -26019.363} C_VEL
LIN {X 0,Y 260.044,Z 850.626,A -85,B 0,C 180,E1 -26022.444,E2 -26022.444} C_VEL
LIN {X 0,Y 261.244,Z 850.207,A -85,B 0,C 180,E1 -26023.964,E2 -26023.964} C_VEL
LIN {X 0,Y 264.376,Z 848.287,A -85,B 0,C 180,E1 -26026.944,E2 -26026.944} C_VEL
LIN {X 0,Y 268.291,Z 844.685,A -85,B 0,C 180,E1 -26029.841,E2 -26029.841} C_VEL
LIN {X 0,Y 271.746,Z 840.932,A -85,B 0,C 180,E1 -26031.947,E2 -26031.947} C_VEL
LIN {X 0,Y 275.746,Z 836.086,A -85,B 0,C 180,E1 -26033.981,E2 -26033.981} C_VEL
LIN {X 0,Y 280.098,Z 830.092,A -85,B 0,C 180,E1 -26035.953,E2 -26035.953} C_VEL
LIN {X 0,Y 284.913,Z 822.784,A -85,B 0,C 180,E1 -26037.847,E2 -26037.847} C_VEL
LIN {X 0,Y 289.344,Z 815.318,A -85,B 0,C 180,E1 -26039.395,E2 -26039.395} C_VEL
LIN {X 0,Y 293.858,Z 806.775,A -85,B 0,C 180,E1 -26040.829,E2 -26040.829} C_VEL
LIN {X 0,Y 298.188,Z 797.668,A -85,B 0,C 180,E1 -26042.074,E2 -26042.074} C_VEL
LIN {X 0,Y 302.142,Z 788.516,A -85,B 0,C 180,E1 -26043.088,E2 -26043.088} C_VEL
LIN {X 0,Y 305.709,Z 779.033,A -85,B 0,C 180,E1 -26043.951,E2 -26043.951} C_VEL
LIN {X 0,Y 309.037,Z 768.689,A -85,B 0,C 180,E1 -26044.714,E2 -26044.714} C_VEL
LIN {X 0,Y 311.889,Z 758.093,A -85,B 0,C 180,E1 -26045.331,E2 -26045.331} C_VEL
LIN {X 0,Y 314.385,Z 746.443,A -85,B 0,C 180,E1 -26045.854,E2 -26045.854} C_VEL
LIN {X 0,Y 319.087,Z 716.832,A -85,B 0,C 180,E1 -26046.965,E2 -26046.965} C_VEL
LIN {X 0,Y 317.29,Z 711.472,A -85,B 0,C 180,E1 -26048.261,E2 -26048.261} C_VEL
LIN {X 0,Y 315.036,Z 705.312,A -85,B 0,C 180,E1 -26050.059,E2 -26050.059} C_VEL
LIN {X 0,Y 313.112,Z 700.885,A -85,B 0,C 180,E1 -26051.755,E2 -26051.755} C_VEL
LIN {X 0,Y 311.362,Z 696.766,A -85,B 0,C 180,E1 -26053.8,E2 -26053.8} C_VEL
LIN {X 0,Y 309.343,Z 691.732,A -85,B 0,C 180,E1 -26057.766,E2 -26057.766} C_VEL
LIN {X 0,Y 308.993,Z 690.916,A -85,B 0,C 180,E1 -26060.6,E2 -26060.6} C_VEL
LIN {X 0,Y 309.442,Z 691.192,A -85,B 0,C 180,E1 -26062.726,E2 -26062.726} C_VEL
LIN {X 0,Y 311.763,Z 694.967,A -85,B 0,C 180,E1 -26066.716,E2 -26066.716} C_VEL
LIN {X 0,Y 313.99,Z 699.229,A -85,B 0,C 180,E1 -26069.067,E2 -26069.067} C_VEL
LIN {X 0,Y 316.066,Z 703.639,A -85,B 0,C 180,E1 -26070.82,E2 -26070.82} C_VEL
LIN {X 0,Y 318.287,Z 708.211,A -85,B 0,C 180,E1 -26072.355,E2 -26072.355} C_VEL
LIN {X 0,Y 319.604,Z 711.53,A -85,B 0,C 180,E1 -26073.248,E2 -26073.248} C_VEL
LIN {X 0,Y 314.317,Z 743.573,A -85,B 0,C 180,E1 -26074.448,E2 -26074.448} C_VEL
LIN {X 0,Y 311.041,Z 757.942,A -85,B 0,C 180,E1 -26075.202,E2 -26075.202} C_VEL
LIN {X 0,Y 307.682,Z 769.31,A -85,B 0,C 180,E1 -26076.012,E2 -26076.012} C_VEL
LIN {X 0,Y 304.123,Z 779.564,A -85,B 0,C 180,E1 -26076.95,E2 -26076.95} C_VEL
LIN {X 0,Y 300.091,Z 789.481,A -85,B 0,C 180,E1 -26078.071,E2 -26078.071} C_VEL
LIN {X 0,Y 296.28,Z 797.806,A -85,B 0,C 180,E1 -26079.23,E2 -26079.23} C_VEL
LIN {X 0,Y 292.597,Z 805.093,A -85,B 0,C 180,E1 -26080.418,E2 -26080.418} C_VEL
LIN {X 0,Y 288.22,Z 812.818,A -85,B 0,C 180,E1 -26081.961,E2 -26081.961} C_VEL
LIN {X 0,Y 284.113,Z 819.246,A -85,B 0,C 180,E1 -26083.529,E2 -26083.529} C_VEL
LIN {X 0,Y 280.972,Z 823.746,A -85,B 0,C 180,E1 -26084.825,E2 -26084.825} C_VEL
LIN {X 0,Y 276.578,Z 829.319,A -85,B 0,C 180,E1 -26086.824,E2 -26086.824} C_VEL
LIN {X 0,Y 272.623,Z 833.725,A -85,B 0,C 180,E1 -26088.889,E2 -26088.889} C_VEL
LIN {X 0,Y 269.051,Z 837.065,A -85,B 0,C 180,E1 -26091.013,E2 -26091.013} C_VEL
LIN {X 0,Y 265.026,Z 839.901,A -85,B 0,C 180,E1 -26093.931,E2 -26093.931} C_VEL
LIN {X 0,Y 263.29,Z 840.799,A -85,B 0,C 180,E1 -26095.422,E2 -26095.422} C_VEL
LIN {X 0,Y 260.62,Z 841.293,A -85,B 0,C 180,E1 -26098.459,E2 -26098.459} C_VEL
LIN {X 0,Y 259.189,Z 840.639,A -85,B 0,C 180,E1 -26100.76,E2 -26100.76} C_VEL
LIN {X 0,Y 258.124,Z 839.062,A -85,B 0,C 180,E1 -26103.111,E2 -26103.111} C_VEL
LIN {X 0,Y 257.261,Z 835.464,A -85,B 0,C 180,E1 -26106.252,E2 -26106.252} C_VEL
LIN {X 0,Y 257.146,Z 831.644,A -85,B 0,C 180,E1 -26108.616,E2 -26108.616} C_VEL
LIN {X 0,Y 257.251,Z 826.674,A -85,B 0,C 180,E1 -26110.987,E2 -26110.987} C_VEL
LIN {X 0,Y 257.449,Z 820.349,A -85,B 0,C 180,E1 -26113.371,E2 -26113.371} C_VEL
LIN {X 0,Y 257.827,Z 813.932,A -85,B 0,C 180,E1 -26115.359,E2 -26115.359} C_VEL
LIN {X 0,Y 258.188,Z 806.039,A -85,B 0,C 180,E1 -26117.362,E2 -26117.362} C_VEL
LIN {X 0,Y 258.713,Z 797.542,A -85,B 0,C 180,E1 -26119.163,E2 -26119.163} C_VEL
LIN {X 0,Y 259.115,Z 789.705,A -85,B 0,C 180,E1 -26120.573,E2 -26120.573} C_VEL
LIN {X 0,Y 259.688,Z 780.5,A -85,B 0,C 180,E1 -26121.977,E2 -26121.977} C_VEL
LIN {X 0,Y 260.4,Z 769.345,A -85,B 0,C 180,E1 -26123.375,E2 -26123.375} C_VEL
LIN {X 0,Y 260.93,Z 759.203,A -85,B 0,C 180,E1 -26124.407,E2 -26124.407} C_VEL
LIN {X 0,Y 261.423,Z 748.651,A -85,B 0,C 180,E1 -26125.267,E2 -26125.267} C_VEL
LIN {X 0,Y 261.772,Z 738.062,A -85,B 0,C 180,E1 -26125.932,E2 -26125.932} C_VEL
LIN {X 0,Y 263.23,Z 696.934,A -85,B 0,C 180,E1 -26127.78,E2 -26127.78} C_VEL
LIN {X 0,Y 264.114,Z 664.116,A -85,B 0,C 180,E1 -26129.2,E2 -26129.2} C_VEL
LIN {X 0,Y 261.468,Z 636.157,A -85,B 0,C 180,E1 -26130.442,E2 -26130.442} C_VEL
LIN {X 0,Y 261.218,Z 629.834,A -85,B 0,C 180,E1 -26130.752,E2 -26130.752} C_VEL
LIN {X 0,Y 260.913,Z 626.44,A -85,B 0,C 180,E1 -26132.06,E2 -26132.06} C_VEL
LIN {X 0,Y 260.607,Z 624.953,A -85,B 0,C 180,E1 -26132.697,E2 -26132.697} C_VEL
LIN {X 0,Y 260.282,Z 624.991,A -85,B 0,C 180,E1 -26136.301,E2 -26136.301} C_VEL
LIN {X 0,Y 260.246,Z 625.001,A -85,B 0,C 180,E1 -26140.236,E2 -26140.236} C_VEL
LIN {X 0,Y 260.238,Z 624.997,A -85,B 0,C 180,E1 -26144.41,E2 -26144.41} C_VEL
LIN {X 0,Y 260.24,Z 624.998,A -85,B 0,C 180,E1 -26148.905,E2 -26148.905} C_VEL
LIN {X 0,Y 260.205,Z 625.006,A -85,B 0,C 180,E1 -26151.747,E2 -26151.747} C_VEL
LIN {X 0,Y 260.223,Z 624.999,A -85,B 0,C 180,E1 -26155.579,E2 -26155.579} C_VEL
LIN {X 0,Y 260.219,Z 625.001,A -85,B 0,C 180,E1 -26159.468,E2 -26159.468} C_VEL
LIN {X 0,Y 260.283,Z 624.992,A -85,B 0,C 180,E1 -26162.775,E2 -26162.775} C_VEL
LIN {X 0,Y 260.295,Z 624.992,A -85,B 0,C 180,E1 -26166.193,E2 -26166.193} C_VEL
LIN {X 0,Y 260.375,Z 624.984,A -85,B 0,C 180,E1 -26170.311,E2 -26170.311} C_VEL
LIN {X 0,Y 260.491,Z 624.964,A -85,B 0,C 180,E1 -26175.467,E2 -26175.467} C_VEL
LIN {X 0,Y 260.491,Z 624.967,A -85,B 0,C 180,E1 -26179.15,E2 -26179.15} C_VEL
LIN {X 0,Y 260.798,Z 624.931,A -85,B 0,C 180,E1 -26183.832,E2 -26183.832} C_VEL
LIN {X 0,Y 260.859,Z 624.923,A -85,B 0,C 180,E1 -26188.461,E2 -26188.461} C_VEL
LIN {X 0,Y 260.981,Z 624.911,A -85,B 0,C 180,E1 -26190,E2 -26190} C_VEL
LIN {X 0,Y 260.8,Z 624.924,A -85,B 0,C 180,E1 -26194.621,E2 -26194.621} C_VEL
LIN {X 0,Y 260.642,Z 624.949,A -85,B 0,C 180,E1 -26197.722,E2 -26197.722} C_VEL
LIN {X 0,Y 260.468,Z 624.969,A -85,B 0,C 180,E1 -26202.423,E2 -26202.423} C_VEL
LIN {X 0,Y 260.388,Z 624.977,A -85,B 0,C 180,E1 -26205.605,E2 -26205.605} C_VEL
LIN {X 0,Y 260.374,Z 624.984,A -85,B 0,C 180,E1 -26209.688,E2 -26209.688} C_VEL
LIN {X 0,Y 260.294,Z 624.992,A -85,B 0,C 180,E1 -26213.806,E2 -26213.806} C_VEL
LIN {X 0,Y 260.272,Z 624.994,A -85,B 0,C 180,E1 -26217.367,E2 -26217.367} C_VEL
LIN {X 0,Y 260.226,Z 625,A -85,B 0,C 180,E1 -26220.758,E2 -26220.758} C_VEL
LIN {X 0,Y 260.261,Z 624.994,A -85,B 0,C 180,E1 -26224.414,E2 -26224.414} C_VEL
LIN {X 0,Y 260.286,Z 624.993,A -85,B 0,C 180,E1 -26228.704,E2 -26228.704} C_VEL
LIN {X 0,Y 260.244,Z 624.997,A -85,B 0,C 180,E1 -26232.289,E2 -26232.289} C_VEL
LIN {X 0,Y 260.24,Z 624.999,A -85,B 0,C 180,E1 -26236.611,E2 -26236.611} C_VEL
LIN {X 0,Y 260.277,Z 624.997,A -85,B 0,C 180,E1 -26239.77,E2 -26239.77} C_VEL
LIN {X 0,Y 260.279,Z 624.992,A -85,B 0,C 180,E1 -26243.836,E2 -26243.836} C_VEL
LIN {X 0,Y 260.233,Z 625,A -85,B 0,C 180,E1 -26247.431,E2 -26247.431} C_VEL
LIN {X 0,Y 260.228,Z 624.998,A -85,B 0,C 180,E1 -26251.021,E2 -26251.021} C_VEL
LIN {X 0,Y 260.267,Z 624.994,A -85,B 0,C 180,E1 -26254.495,E2 -26254.495} C_VEL
LIN {X 0,Y 260.303,Z 624.994,A -85,B 0,C 180,E1 -26257.87,E2 -26257.87} C_VEL
LIN {X 0,Y 260.353,Z 624.983,A -85,B 0,C 180,E1 -26261.166,E2 -26261.166} C_VEL
LIN {X 0,Y 260.451,Z 624.975,A -85,B 0,C 180,E1 -26265.994,E2 -26265.994} C_VEL
LIN {X 0,Y 260.561,Z 624.957,A -85,B 0,C 180,E1 -26270.719,E2 -26270.719} C_VEL
LIN {X 0,Y 260.801,Z 624.927,A -85,B 0,C 180,E1 -26273.833,E2 -26273.833} C_VEL
LIN {X 0,Y 260.863,Z 624.922,A -85,B 0,C 180,E1 -26278.462,E2 -26278.462} C_VEL
LIN {X 0,Y 260.982,Z 624.908,A -85,B 0,C 180,E1 -26280,E2 -26280} C_VEL
LIN {X 0,Y 260.802,Z 624.928,A -85,B 0,C 180,E1 -26284.622,E2 -26284.622} C_VEL
LIN {X 0,Y 260.645,Z 624.951,A -85,B 0,C 180,E1 -26287.723,E2 -26287.723} C_VEL
LIN {X 0,Y 260.431,Z 624.973,A -85,B 0,C 180,E1 -26292.426,E2 -26292.426} C_VEL
LIN {X 0,Y 260.344,Z 624.986,A -85,B 0,C 180,E1 -26295.608,E2 -26295.608} C_VEL
LIN {X 0,Y 260.311,Z 624.991,A -85,B 0,C 180,E1 -26299.648,E2 -26299.648} C_VEL
LIN {X 0,Y 260.298,Z 624.991,A -85,B 0,C 180,E1 -26303.806,E2 -26303.806} C_VEL
LIN {X 0,Y 260.276,Z 624.995,A -85,B 0,C 180,E1 -26307.367,E2 -26307.367} C_VEL
LIN {X 0,Y 260.206,Z 624.999,A -85,B 0,C 180,E1 -26310.761,E2 -26310.761} C_VEL
LIN {X 0,Y 260.223,Z 625.002,A -85,B 0,C 180,E1 -26314.421,E2 -26314.421} C_VEL
LIN {X 0,Y 260.216,Z 625.001,A -85,B 0,C 180,E1 -26318.683,E2 -26318.683} C_VEL
LIN {X 0,Y 260.203,Z 625.003,A -85,B 0,C 180,E1 -26322.298,E2 -26322.298} C_VEL
LIN {X 0,Y 260.19,Z 625.005,A -85,B 0,C 180,E1 -26326.624,E2 -26326.624} C_VEL
LIN {X 0,Y 260.237,Z 625,A -85,B 0,C 180,E1 -26329.762,E2 -26329.762} C_VEL
LIN {X 0,Y 260.229,Z 625.002,A -85,B 0,C 180,E1 -26333.852,E2 -26333.852} C_VEL
LIN {X 0,Y 260.224,Z 625.001,A -85,B 0,C 180,E1 -26337.43,E2 -26337.43} C_VEL
LIN {X 0,Y 260.505,Z 624.983,A -85,B 0,C 180,E1 -26343.179,E2 -26343.179} C_VEL
LIN {X 0,Y 262.043,Z 633.62,A -85,B 0,C 180,E1 -26346.363,E2 -26346.363} C_VEL
LIN {X 0,Y 260.757,Z 641.706,A -85,B 0,C 180,E1 -26349.253,E2 -26349.253} C_VEL
LIN {X 0,Y 261.461,Z 661.199,A -85,B 0,C 180,E1 -26350.118,E2 -26350.118} C_VEL
LIN {X 0,Y 263.766,Z 689.606,A -85,B 0,C 180,E1 -26351.371,E2 -26351.371} C_VEL
LIN {X 0,Y 263.639,Z 694.162,A -85,B 0,C 180,E1 -26351.567,E2 -26351.567} C_VEL
LIN {X 0,Y 262.719,Z 699.893,A -85,B 0,C 180,E1 -26351.813,E2 -26351.813} C_VEL
LIN {X 0,Y 256.536,Z 718.352,A -85,B 0,C 180,E1 -26352.642,E2 -26352.642} C_VEL
LIN {X 0,Y 255.695,Z 724.082,A -85,B 0,C 180,E1 -26352.904,E2 -26352.904} C_VEL
LIN {X 0,Y 254.846,Z 750.58,A -85,B 0,C 180,E1 -26354.169,E2 -26354.169} C_VEL
LIN {X 0,Y 254.305,Z 763.668,A -85,B 0,C 180,E1 -26355.059,E2 -26355.059} C_VEL
LIN {X 0,Y 253.741,Z 776.212,A -85,B 0,C 180,E1 -26356.226,E2 -26356.226} C_VEL
LIN {X 0,Y 253.06,Z 787.713,A -85,B 0,C 180,E1 -26357.613,E2 -26357.613} C_VEL
LIN {X 0,Y 252.516,Z 797.208,A -85,B 0,C 180,E1 -26359.006,E2 -26359.006} C_VEL
LIN {X 0,Y 251.982,Z 806.277,A -85,B 0,C 180,E1 -26360.601,E2 -26360.601} C_VEL
LIN {X 0,Y 251.524,Z 814.823,A -85,B 0,C 180,E1 -26362.399,E2 -26362.399} C_VEL
LIN {X 0,Y 251.345,Z 821.303,A -85,B 0,C 180,E1 -26364.002,E2 -26364.002} C_VEL
LIN {X 0,Y 251.153,Z 828.079,A -85,B 0,C 180,E1 -26366.002,E2 -26366.002} C_VEL
LIN {X 0,Y 251.088,Z 832.735,A -85,B 0,C 180,E1 -26367.602,E2 -26367.602} C_VEL
LIN {X 0,Y 250.857,Z 838.38,A -85,B 0,C 180,E1 -26370,E2 -26370} C_VEL
LIN {X 0,Y 250.62,Z 842.776,A -85,B 0,C 180,E1 -26372.403,E2 -26372.403} C_VEL
LIN {X 0,Y 250.514,Z 846.09,A -85,B 0,C 180,E1 -26374.812,E2 -26374.812} C_VEL
LIN {X 0,Y 250.799,Z 848.956,A -85,B 0,C 180,E1 -26378.027,E2 -26378.027} C_VEL
LIN {X 0,Y 252.146,Z 850.297,A -85,B 0,C 180,E1 -26381.213,E2 -26381.213} C_VEL
LIN {X 0,Y 253.105,Z 850.508,A -85,B 0,C 180,E1 -26382.791,E2 -26382.791} C_VEL
LIN {X 0,Y 255.87,Z 849.598,A -85,B 0,C 180,E1 -26385.888,E2 -26385.888} C_VEL
LIN {X 0,Y 259.482,Z 847.139,A -85,B 0,C 180,E1 -26388.901,E2 -26388.901} C_VEL
LIN {X 0,Y 261.668,Z 845.415,A -85,B 0,C 180,E1 -26390.365,E2 -26390.365} C_VEL
LIN {X 0,Y 266.545,Z 840.468,A -85,B 0,C 180,E1 -26393.215,E2 -26393.215} C_VEL
LIN {X 0,Y 270.836,Z 835.643,A -85,B 0,C 180,E1 -26395.26,E2 -26395.26} C_VEL
LIN {X 0,Y 275.5,Z 829.641,A -85,B 0,C 180,E1 -26397.235,E2 -26397.235} C_VEL
LIN {X 0,Y 280.565,Z 822.259,A -85,B 0,C 180,E1 -26399.133,E2 -26399.133} C_VEL
LIN {X 0,Y 285.171,Z 814.898,A -85,B 0,C 180,E1 -26400.642,E2 -26400.642} C_VEL
LIN {X 0,Y 289.027,Z 808.186,A -85,B 0,C 180,E1 -26401.81,E2 -26401.81} C_VEL
LIN {X 0,Y 294.127,Z 798.122,A -85,B 0,C 180,E1 -26403.212,E2 -26403.212} C_VEL
LIN {X 0,Y 298.468,Z 788.441,A -85,B 0,C 180,E1 -26404.28,E2 -26404.28} C_VEL
LIN {X 0,Y 302.402,Z 778.302,A -85,B 0,C 180,E1 -26405.182,E2 -26405.182} C_VEL
LIN {X 0,Y 306.465,Z 765.951,A -85,B 0,C 180,E1 -26406.053,E2 -26406.053} C_VEL
LIN {X 0,Y 309.395,Z 755.112,A -85,B 0,C 180,E1 -26406.652,E2 -26406.652} C_VEL
LIN {X 0,Y 312.37,Z 740.745,A -85,B 0,C 180,E1 -26407.261,E2 -26407.261} C_VEL
LIN {X 0,Y 315.624,Z 720.414,A -85,B 0,C 180,E1 -26408.018,E2 -26408.018} C_VEL
LIN {X 0,Y 313.385,Z 713.665,A -85,B 0,C 180,E1 -26409.841,E2 -26409.841} C_VEL
LIN {X 0,Y 311.926,Z 709.747,A -85,B 0,C 180,E1 -26411.184,E2 -26411.184} C_VEL
LIN {X 0,Y 310.898,Z 707.114,A -85,B 0,C 180,E1 -26412.239,E2 -26412.239} C_VEL
LIN {X 0,Y 309.401,Z 703.319,A -85,B 0,C 180,E1 -26414.138,E2 -26414.138} C_VEL
LIN {X 0,Y 307.68,Z 698.588,A -85,B 0,C 180,E1 -26417.923,E2 -26417.923} C_VEL
LIN {X 0,Y 307.4,Z 697.826,A -85,B 0,C 180,E1 -26420.781,E2 -26420.781} C_VEL
LIN {X 0,Y 307.866,Z 698.233,A -85,B 0,C 180,E1 -26422.944,E2 -26422.944} C_VEL
LIN {X 0,Y 309.955,Z 701.873,A -85,B 0,C 180,E1 -26426.583,E2 -26426.583} C_VEL
LIN {X 0,Y 311.901,Z 705.938,A -85,B 0,C 180,E1 -26428.795,E2 -26428.795} C_VEL
LIN {X 0,Y 313.812,Z 710.098,A -85,B 0,C 180,E1 -26430.461,E2 -26430.461} C_VEL
LIN {X 0,Y 315.735,Z 714.461,A -85,B 0,C 180,E1 -26431.926,E2 -26431.926} C_VEL
LIN {X 0,Y 316.139,Z 715.621,A -85,B 0,C 180,E1 -26432.225,E2 -26432.225} C_VEL
LIN {X 0,Y 311.428,Z 742.878,A -85,B 0,C 180,E1 -26433.231,E2 -26433.231} C_VEL
LIN {X 0,Y 308.113,Z 757.086,A -85,B 0,C 180,E1 -26433.957,E2 -26433.957} C_VEL
LIN {X 0,Y 304.35,Z 769.151,A -85,B 0,C 180,E1 -26434.8,E2 -26434.8} C_VEL
LIN {X 0,Y 300.698,Z 779.363,A -85,B 0,C 180,E1 -26435.722,E2 -26435.722} C_VEL
LIN {X 0,Y 296.909,Z 788.495,A -85,B 0,C 180,E1 -26436.724,E2 -26436.724} C_VEL
LIN {X 0,Y 292.868,Z 797.056,A -85,B 0,C 180,E1 -26437.871,E2 -26437.871} C_VEL
LIN {X 0,Y 288.936,Z 804.436,A -85,B 0,C 180,E1 -26439.048,E2 -26439.048} C_VEL
LIN {X 0,Y 284.334,Z 812.161,A -85,B 0,C 180,E1 -26440.575,E2 -26440.575} C_VEL
LIN {X 0,Y 279.963,Z 818.826,A -85,B 0,C 180,E1 -26442.165,E2 -26442.165} C_VEL
LIN {X 0,Y 275.821,Z 824.399,A -85,B 0,C 180,E1 -26443.779,E2 -26443.779} C_VEL
LIN {X 0,Y 271.166,Z 829.848,A -85,B 0,C 180,E1 -26445.795,E2 -26445.795} C_VEL
LIN {X 0,Y 266.945,Z 834.147,A -85,B 0,C 180,E1 -26447.882,E2 -26447.882} C_VEL
LIN {X 0,Y 263.08,Z 837.516,A -85,B 0,C 180,E1 -26450.104,E2 -26450.104} C_VEL
LIN {X 0,Y 259.867,Z 839.737,A -85,B 0,C 180,E1 -26452.254,E2 -26452.254} C_VEL
LIN {X 0,Y 256.159,Z 841.281,A -85,B 0,C 180,E1 -26455.294,E2 -26455.294} C_VEL
LIN {X 0,Y 254.723,Z 841.507,A -85,B 0,C 180,E1 -26456.847,E2 -26456.847} C_VEL
LIN {X 0,Y 252.46,Z 840.787,A -85,B 0,C 180,E1 -26459.999,E2 -26459.999} C_VEL
LIN {X 0,Y 250.989,Z 838.38,A -85,B 0,C 180,E1 -26463.199,E2 -26463.199} C_VEL
LIN {X 0,Y 250.303,Z 835.567,A -85,B 0,C 180,E1 -26465.62,E2 -26465.62} C_VEL
LIN {X 0,Y 250.075,Z 831.733,A -85,B 0,C 180,E1 -26468.05,E2 -26468.05} C_VEL
LIN {X 0,Y 250.207,Z 826.76,A -85,B 0,C 180,E1 -26470.484,E2 -26470.484} C_VEL
LIN {X 0,Y 250.401,Z 820.429,A -85,B 0,C 180,E1 -26472.931,E2 -26472.931} C_VEL
LIN {X 0,Y 250.781,Z 814.026,A -85,B 0,C 180,E1 -26474.972,E2 -26474.972} C_VEL
LIN {X 0,Y 251.104,Z 806.206,A -85,B 0,C 180,E1 -26477.031,E2 -26477.031} C_VEL
LIN {X 0,Y 251.596,Z 798.152,A -85,B 0,C 180,E1 -26478.814,E2 -26478.814} C_VEL
LIN {X 0,Y 252.029,Z 790.049,A -85,B 0,C 180,E1 -26480.328,E2 -26480.328} C_VEL
LIN {X 0,Y 252.577,Z 780.873,A -85,B 0,C 180,E1 -26481.771,E2 -26481.771} C_VEL
LIN {X 0,Y 253.255,Z 769.772,A -85,B 0,C 180,E1 -26483.207,E2 -26483.207} C_VEL
LIN {X 0,Y 253.853,Z 759.257,A -85,B 0,C 180,E1 -26484.31,E2 -26484.31} C_VEL
LIN {X 0,Y 254.313,Z 749.128,A -85,B 0,C 180,E1 -26485.162,E2 -26485.162} C_VEL
LIN {X 0,Y 254.666,Z 738.893,A -85,B 0,C 180,E1 -26485.834,E2 -26485.834} C_VEL
LIN {X 0,Y 255.664,Z 711.011,A -85,B 0,C 180,E1 -26487.15,E2 -26487.15} C_VEL
LIN {X 0,Y 257.09,Z 664.971,A -85,B 0,C 180,E1 -26489.221,E2 -26489.221} C_VEL
LIN {X 0,Y 254.402,Z 636.428,A -85,B 0,C 180,E1 -26490.536,E2 -26490.536} C_VEL
LIN {X 0,Y 254.139,Z 629.994,A -85,B 0,C 180,E1 -26490.867,E2 -26490.867} C_VEL
LIN {X 0,Y 253.572,Z 625.83,A -85,B 0,C 180,E1 -26492.532,E2 -26492.532} C_VEL
LIN {X 0,Y 253.177,Z 625.875,A -85,B 0,C 180,E1 -26497.492,E2 -26497.492} C_VEL
LIN {X 0,Y 253.17,Z 625.881,A -85,B 0,C 180,E1 -26501.668,E2 -26501.668} C_VEL
LIN {X 0,Y 253.177,Z 625.877,A -85,B 0,C 180,E1 -26505.997,E2 -26505.997} C_VEL
LIN {X 0,Y 253.167,Z 625.881,A -85,B 0,C 180,E1 -26510.48,E2 -26510.48} C_VEL
LIN {X 0,Y 253.169,Z 625.877,A -85,B 0,C 180,E1 -26514.478,E2 -26514.478} C_VEL
LIN {X 0,Y 253.165,Z 625.882,A -85,B 0,C 180,E1 -26518.285,E2 -26518.285} C_VEL
LIN {X 0,Y 253.218,Z 625.875,A -85,B 0,C 180,E1 -26522.271,E2 -26522.271} C_VEL
LIN {X 0,Y 253.238,Z 625.869,A -85,B 0,C 180,E1 -26525.888,E2 -26525.888} C_VEL
LIN {X 0,Y 253.345,Z 625.858,A -85,B 0,C 180,E1 -26530.623,E2 -26530.623} C_VEL
LIN {X 0,Y 253.449,Z 625.841,A -85,B 0,C 180,E1 -26535.597,E2 -26535.597} C_VEL
LIN {X 0,Y 253.509,Z 625.838,A -85,B 0,C 180,E1 -26540.457,E2 -26540.457} C_VEL
LIN {X 0,Y 253.748,Z 625.808,A -85,B 0,C 180,E1 -26543.66,E2 -26543.66} C_VEL
LIN {X 0,Y 253.814,Z 625.8,A -85,B 0,C 180,E1 -26548.418,E2 -26548.418} C_VEL
LIN {X 0,Y 253.942,Z 625.788,A -85,B 0,C 180,E1 -26550,E2 -26550} C_VEL
LIN {X 0,Y 253.747,Z 625.802,A -85,B 0,C 180,E1 -26554.75,E2 -26554.75} C_VEL
LIN {X 0,Y 253.575,Z 625.831,A -85,B 0,C 180,E1 -26557.938,E2 -26557.938} C_VEL
LIN {X 0,Y 253.425,Z 625.845,A -85,B 0,C 180,E1 -26562.774,E2 -26562.774} C_VEL
LIN {X 0,Y 253.326,Z 625.861,A -85,B 0,C 180,E1 -26566.051,E2 -26566.051} C_VEL
LIN {X 0,Y 253.321,Z 625.865,A -85,B 0,C 180,E1 -26569.931,E2 -26569.931} C_VEL
LIN {X 0,Y 253.226,Z 625.869,A -85,B 0,C 180,E1 -26574.514,E2 -26574.514} C_VEL
LIN {X 0,Y 253.202,Z 625.879,A -85,B 0,C 180,E1 -26578.052,E2 -26578.052} C_VEL
LIN {X 0,Y 253.178,Z 625.88,A -85,B 0,C 180,E1 -26581.712,E2 -26581.712} C_VEL
LIN {X 0,Y 253.218,Z 625.871,A -85,B 0,C 180,E1 -26585.513,E2 -26585.513} C_VEL
LIN {X 0,Y 253.223,Z 625.874,A -85,B 0,C 180,E1 -26589.509,E2 -26589.509} C_VEL
LIN {X 0,Y 253.187,Z 625.876,A -85,B 0,C 180,E1 -26593.759,E2 -26593.759} C_VEL
LIN {X 0,Y 253.222,Z 625.874,A -85,B 0,C 180,E1 -26598.405,E2 -26598.405} C_VEL
LIN {X 0,Y 253.201,Z 625.872,A -85,B 0,C 180,E1 -26602.513,E2 -26602.513} C_VEL
LIN {X 0,Y 253.22,Z 625.874,A -85,B 0,C 180,E1 -26606.412,E2 -26606.412} C_VEL
LIN {X 0,Y 253.156,Z 625.883,A -85,B 0,C 180,E1 -26610.131,E2 -26610.131} C_VEL
LIN {X 0,Y 253.216,Z 625.871,A -85,B 0,C 180,E1 -26613.731,E2 -26613.731} C_VEL
LIN {X 0,Y 253.229,Z 625.872,A -85,B 0,C 180,E1 -26617.217,E2 -26617.217} C_VEL
LIN {X 0,Y 253.333,Z 625.858,A -85,B 0,C 180,E1 -26620.623,E2 -26620.623} C_VEL
LIN {X 0,Y 253.424,Z 625.847,A -85,B 0,C 180,E1 -26625.597,E2 -26625.597} C_VEL
LIN {X 0,Y 253.509,Z 625.836,A -85,B 0,C 180,E1 -26630.458,E2 -26630.458} C_VEL
LIN {X 0,Y 253.778,Z 625.801,A -85,B 0,C 180,E1 -26633.662,E2 -26633.662} C_VEL
LIN {X 0,Y 253.818,Z 625.8,A -85,B 0,C 180,E1 -26638.419,E2 -26638.419} C_VEL
LIN {X 0,Y 253.943,Z 625.785,A -85,B 0,C 180,E1 -26640.001,E2 -26640.001} C_VEL
LIN {X 0,Y 253.749,Z 625.806,A -85,B 0,C 180,E1 -26644.751,E2 -26644.751} C_VEL
LIN {X 0,Y 253.578,Z 625.833,A -85,B 0,C 180,E1 -26647.939,E2 -26647.939} C_VEL
LIN {X 0,Y 253.382,Z 625.849,A -85,B 0,C 180,E1 -26652.777,E2 -26652.777} C_VEL
LIN {X 0,Y 253.289,Z 625.869,A -85,B 0,C 180,E1 -26656.054,E2 -26656.054} C_VEL
LIN {X 0,Y 253.243,Z 625.872,A -85,B 0,C 180,E1 -26659.881,E2 -26659.881} C_VEL
LIN {X 0,Y 253.229,Z 625.872,A -85,B 0,C 180,E1 -26664.514,E2 -26664.514} C_VEL
LIN {X 0,Y 253.203,Z 625.878,A -85,B 0,C 180,E1 -26668.053,E2 -26668.053} C_VEL
LIN {X 0,Y 253.16,Z 625.879,A -85,B 0,C 180,E1 -26671.715,E2 -26671.715} C_VEL
LIN {X 0,Y 253.169,Z 625.88,A -85,B 0,C 180,E1 -26675.522,E2 -26675.522} C_VEL
LIN {X 0,Y 253.164,Z 625.88,A -85,B 0,C 180,E1 -26679.521,E2 -26679.521} C_VEL
LIN {X 0,Y 253.129,Z 625.885,A -85,B 0,C 180,E1 -26683.772,E2 -26683.772} C_VEL
LIN {X 0,Y 253.166,Z 625.88,A -85,B 0,C 180,E1 -26688.393,E2 -26688.393} C_VEL
LIN {X 0,Y 253.137,Z 625.883,A -85,B 0,C 180,E1 -26692.501,E2 -26692.501} C_VEL
LIN {X 0,Y 253.211,Z 625.876,A -85,B 0,C 180,E1 -26696.41,E2 -26696.41} C_VEL
LIN {X 0,Y 253.176,Z 625.877,A -85,B 0,C 180,E1 -26700.133,E2 -26700.133} C_VEL
LIN {X 0,Y 253.496,Z 626,A -85,B 0,C 180,E1 -26703.32,E2 -26703.32} C_VEL
LIN {X 0,Y 254.877,Z 633.294,A -85,B 0,C 180,E1 -26706.087,E2 -26706.087} C_VEL
LIN {X 0,Y 254.128,Z 638.9,A -85,B 0,C 180,E1 -26708.155,E2 -26708.155} C_VEL
LIN {X 0,Y 253.691,Z 641.565,A -85,B 0,C 180,E1 -26709.139,E2 -26709.139} C_VEL
LIN {X 0,Y 254.313,Z 660.394,A -85,B 0,C 180,E1 -26710.009,E2 -26710.009} C_VEL
LIN {X 0,Y 256.689,Z 689.663,A -85,B 0,C 180,E1 -26711.351,E2 -26711.351} C_VEL
LIN {X 0,Y 255.695,Z 724.082,A -85,B 0,C 180,E1 -26712.904,E2 -26712.904} C_VEL
LIN {X 0,Y 254.844,Z 727.916,A -85,B 0,C 180,E1 -26713.079,E2 -26713.079} C_VEL
LIN {X 0,Y 248.685,Z 739.687,A -85,B 0,C 180,E1 -26713.668,E2 -26713.668} C_VEL
LIN {X 0,Y 248.04,Z 743.512,A -85,B 0,C 180,E1 -26713.856,E2 -26713.856} C_VEL
LIN {X 0,Y 247.444,Z 757.211,A -85,B 0,C 180,E1 -26714.683,E2 -26714.683} C_VEL
LIN {X 0,Y 246.981,Z 768.704,A -85,B 0,C 180,E1 -26715.632,E2 -26715.632} C_VEL
LIN {X 0,Y 246.534,Z 778.526,A -85,B 0,C 180,E1 -26716.654,E2 -26716.654} C_VEL
LIN {X 0,Y 245.922,Z 788.135,A -85,B 0,C 180,E1 -26717.875,E2 -26717.875} C_VEL
LIN {X 0,Y 245.405,Z 797.456,A -85,B 0,C 180,E1 -26719.309,E2 -26719.309} C_VEL
LIN {X 0,Y 244.924,Z 806.386,A -85,B 0,C 180,E1 -26720.951,E2 -26720.951} C_VEL
LIN {X 0,Y 244.54,Z 813.963,A -85,B 0,C 180,E1 -26722.595,E2 -26722.595} C_VEL
LIN {X 0,Y 244.357,Z 820.528,A -85,B 0,C 180,E1 -26724.242,E2 -26724.242} C_VEL
LIN {X 0,Y 244.174,Z 827.398,A -85,B 0,C 180,E1 -26726.3,E2 -26726.3} C_VEL
LIN {X 0,Y 244.065,Z 833.128,A -85,B 0,C 180,E1 -26728.356,E2 -26728.356} C_VEL
LIN {X 0,Y 243.874,Z 838.622,A -85,B 0,C 180,E1 -26730.823,E2 -26730.823} C_VEL
LIN {X 0,Y 243.561,Z 842.872,A -85,B 0,C 180,E1 -26733.298,E2 -26733.298} C_VEL
LIN {X 0,Y 243.519,Z 846.818,A -85,B 0,C 180,E1 -26736.607,E2 -26736.607} C_VEL
LIN {X 0,Y 243.788,Z 848.301,A -85,B 0,C 180,E1 -26738.26,E2 -26738.26} C_VEL
LIN {X 0,Y 245.198,Z 849.993,A -85,B 0,C 180,E1 -26741.535,E2 -26741.535} C_VEL
LIN {X 0,Y 247.508,Z 850.12,A -85,B 0,C 180,E1 -26744.756,E2 -26744.756} C_VEL
LIN {X 0,Y 249.055,Z 849.701,A -85,B 0,C 180,E1 -26746.335,E2 -26746.335} C_VEL
LIN {X 0,Y 252.806,Z 847.649,A -85,B 0,C 180,E1 -26749.42,E2 -26749.42} C_VEL
LIN {X 0,Y 257.462,Z 843.936,A -85,B 0,C 180,E1 -26752.389,E2 -26752.389} C_VEL
LIN {X 0,Y 261.556,Z 840.128,A -85,B 0,C 180,E1 -26754.525,E2 -26754.525} C_VEL
LIN {X 0,Y 266.107,Z 835.255,A -85,B 0,C 180,E1 -26756.582,E2 -26756.582} C_VEL
LIN {X 0,Y 271.041,Z 829.186,A -85,B 0,C 180,E1 -26758.561,E2 -26758.561} C_VEL
LIN {X 0,Y 275.5,Z 823.246,A -85,B 0,C 180,E1 -26760.141,E2 -26760.141} C_VEL
LIN {X 0,Y 280.288,Z 816.179,A -85,B 0,C 180,E1 -26761.655,E2 -26761.655} C_VEL
LIN {X 0,Y 285.318,Z 807.769,A -85,B 0,C 180,E1 -26763.109,E2 -26763.109} C_VEL
LIN {X 0,Y 290.091,Z 798.758,A -85,B 0,C 180,E1 -26764.361,E2 -26764.361} C_VEL
LIN {X 0,Y 295.161,Z 788.021,A -85,B 0,C 180,E1 -26765.55,E2 -26765.55} C_VEL
LIN {X 0,Y 299.291,Z 777.973,A -85,B 0,C 180,E1 -26766.432,E2 -26766.432} C_VEL
LIN {X 0,Y 302.87,Z 767.649,A -85,B 0,C 180,E1 -26767.171,E2 -26767.171} C_VEL
LIN {X 0,Y 305.611,Z 758.294,A -85,B 0,C 180,E1 -26767.71,E2 -26767.71} C_VEL
LIN {X 0,Y 308.419,Z 746.393,A -85,B 0,C 180,E1 -26768.239,E2 -26768.239} C_VEL
LIN {X 0,Y 312.275,Z 724.088,A -85,B 0,C 180,E1 -26769.091,E2 -26769.091} C_VEL
LIN {X 0,Y 310.271,Z 717.606,A -85,B 0,C 180,E1 -26771.029,E2 -26771.029} C_VEL
LIN {X 0,Y 308.707,Z 713.292,A -85,B 0,C 180,E1 -26772.756,E2 -26772.756} C_VEL
LIN {X 0,Y 307.41,Z 709.871,A -85,B 0,C 180,E1 -26774.496,E2 -26774.496} C_VEL
LIN {X 0,Y 306.01,Z 705.446,A -85,B 0,C 180,E1 -26778.068,E2 -26778.068} C_VEL
LIN {X 0,Y 305.71,Z 704.746,A -85,B 0,C 180,E1 -26780.093,E2 -26780.093} C_VEL
LIN {X 0,Y 306.19,Z 705.158,A -85,B 0,C 180,E1 -26782.842,E2 -26782.842} C_VEL
LIN {X 0,Y 308.053,Z 708.654,A -85,B 0,C 180,E1 -26786.349,E2 -26786.349} C_VEL
LIN {X 0,Y 309.718,Z 712.291,A -85,B 0,C 180,E1 -26788.368,E2 -26788.368} C_VEL
LIN {X 0,Y 311.489,Z 716.332,A -85,B 0,C 180,E1 -26790.021,E2 -26790.021} C_VEL
LIN {X 0,Y 312.794,Z 719.658,A -85,B 0,C 180,E1 -26791.167,E2 -26791.167} C_VEL
LIN {X 0,Y 308.451,Z 743.634,A -85,B 0,C 180,E1 -26792.051,E2 -26792.051} C_VEL
LIN {X 0,Y 304.762,Z 758.528,A -85,B 0,C 180,E1 -26792.819,E2 -26792.819} C_VEL
LIN {X 0,Y 301.151,Z 769.64,A -85,B 0,C 180,E1 -26793.587,E2 -26793.587} C_VEL
LIN {X 0,Y 297.216,Z 779.99,A -85,B 0,C 180,E1 -26794.526,E2 -26794.526} C_VEL
LIN {X 0,Y 293.251,Z 788.959,A -85,B 0,C 180,E1 -26795.521,E2 -26795.521} C_VEL
LIN {X 0,Y 288.587,Z 798.233,A -85,B 0,C 180,E1 -26796.77,E2 -26796.77} C_VEL
LIN {X 0,Y 284.515,Z 805.489,A -85,B 0,C 180,E1 -26797.948,E2 -26797.948} C_VEL
LIN {X 0,Y 279.706,Z 813.119,A -85,B 0,C 180,E1 -26799.476,E2 -26799.476} C_VEL
LIN {X 0,Y 274.943,Z 819.774,A -85,B 0,C 180,E1 -26801.119,E2 -26801.119} C_VEL
LIN {X 0,Y 270.764,Z 825.027,A -85,B 0,C 180,E1 -26802.692,E2 -26802.692} C_VEL
LIN {X 0,Y 265.869,Z 830.414,A -85,B 0,C 180,E1 -26804.724,E2 -26804.724} C_VEL
LIN {X 0,Y 261.393,Z 834.642,A -85,B 0,C 180,E1 -26806.834,E2 -26806.834} C_VEL
LIN {X 0,Y 257.403,Z 837.821,A -85,B 0,C 180,E1 -26809.019,E2 -26809.019} C_VEL
LIN {X 0,Y 252.776,Z 840.511,A -85,B 0,C 180,E1 -26812.036,E2 -26812.036} C_VEL
LIN {X 0,Y 250.799,Z 841.369,A -85,B 0,C 180,E1 -26813.585,E2 -26813.585} C_VEL
LIN {X 0,Y 247.583,Z 841.657,A -85,B 0,C 180,E1 -26816.756,E2 -26816.756} C_VEL
LIN {X 0,Y 246.345,Z 841.236,A -85,B 0,C 180,E1 -26818.37,E2 -26818.37} C_VEL
LIN {X 0,Y 244.503,Z 839.296,A -85,B 0,C 180,E1 -26821.641,E2 -26821.641} C_VEL
LIN {X 0,Y 243.417,Z 835.609,A -85,B 0,C 180,E1 -26824.952,E2 -26824.952} C_VEL
LIN {X 0,Y 243.068,Z 831.766,A -85,B 0,C 180,E1 -26827.45,E2 -26827.45} C_VEL
LIN {X 0,Y 243.15,Z 826.834,A -85,B 0,C 180,E1 -26829.953,E2 -26829.953} C_VEL
LIN {X 0,Y 243.364,Z 820.754,A -85,B 0,C 180,E1 -26832.381,E2 -26832.381} C_VEL
LIN {X 0,Y 243.711,Z 814.087,A -85,B 0,C 180,E1 -26834.565,E2 -26834.565} C_VEL
LIN {X 0,Y 244.065,Z 806.279,A -85,B 0,C 180,E1 -26836.677,E2 -26836.677} C_VEL
LIN {X 0,Y 244.547,Z 797.78,A -85,B 0,C 180,E1 -26838.598,E2 -26838.598} C_VEL
LIN {X 0,Y 245.026,Z 788.905,A -85,B 0,C 180,E1 -26840.28,E2 -26840.28} C_VEL
LIN {X 0,Y 245.564,Z 779.578,A -85,B 0,C 180,E1 -26841.765,E2 -26841.765} C_VEL
LIN {X 0,Y 246.15,Z 770.078,A -85,B 0,C 180,E1 -26843.033,E2 -26843.033} C_VEL
LIN {X 0,Y 246.755,Z 759.785,A -85,B 0,C 180,E1 -26844.162,E2 -26844.162} C_VEL
LIN {X 0,Y 247.217,Z 749.356,A -85,B 0,C 180,E1 -26845.07,E2 -26845.07} C_VEL
LIN {X 0,Y 247.595,Z 737.796,A -85,B 0,C 180,E1 -26845.838,E2 -26845.838} C_VEL
LIN {X 0,Y 249.487,Z 682.74,A -85,B 0,C 180,E1 -26848.45,E2 -26848.45} C_VEL
LIN {X 0,Y 249.924,Z 665.049,A -85,B 0,C 180,E1 -26849.27,E2 -26849.27} C_VEL
LIN {X 0,Y 247.349,Z 637.179,A -85,B 0,C 180,E1 -26850.597,E2 -26850.597} C_VEL
LIN {X 0,Y 247.064,Z 630.186,A -85,B 0,C 180,E1 -26850.961,E2 -26850.961} C_VEL
LIN {X 0,Y 246.563,Z 626.703,A -85,B 0,C 180,E1 -26852.447,E2 -26852.447} C_VEL
LIN {X 0,Y 246.144,Z 626.75,A -85,B 0,C 180,E1 -26857.175,E2 -26857.175} C_VEL
LIN {X 0,Y 246.103,Z 626.76,A -85,B 0,C 180,E1 -26860.889,E2 -26860.889} C_VEL
LIN {X 0,Y 246.115,Z 626.755,A -85,B 0,C 180,E1 -26865.356,E2 -26865.356} C_VEL
LIN {X 0,Y 246.094,Z 626.76,A -85,B 0,C 180,E1 -26869.107,E2 -26869.107} C_VEL
LIN {X 0,Y 246.105,Z 626.759,A -85,B 0,C 180,E1 -26873.295,E2 -26873.295} C_VEL
LIN {X 0,Y 246.113,Z 626.755,A -85,B 0,C 180,E1 -26877.265,E2 -26877.265} C_VEL
LIN {X 0,Y 246.163,Z 626.756,A -85,B 0,C 180,E1 -26881.894,E2 -26881.894} C_VEL
LIN {X 0,Y 246.185,Z 626.747,A -85,B 0,C 180,E1 -26886.526,E2 -26886.526} C_VEL
LIN {X 0,Y 246.273,Z 626.743,A -85,B 0,C 180,E1 -26890.043,E2 -26890.043} C_VEL
LIN {X 0,Y 246.389,Z 626.719,A -85,B 0,C 180,E1 -26895.175,E2 -26895.175} C_VEL
LIN {X 0,Y 246.439,Z 626.721,A -85,B 0,C 180,E1 -26900.181,E2 -26900.181} C_VEL
LIN {X 0,Y 246.702,Z 626.685,A -85,B 0,C 180,E1 -26903.572,E2 -26903.572} C_VEL
LIN {X 0,Y 246.76,Z 626.676,A -85,B 0,C 180,E1 -26906.745,E2 -26906.745} C_VEL
LIN {X 0,Y 246.905,Z 626.664,A -85,B 0,C 180,E1 -26910,E2 -26910} C_VEL
LIN {X 0,Y 246.694,Z 626.681,A -85,B 0,C 180,E1 -26914.886,E2 -26914.886} C_VEL
LIN {X 0,Y 246.518,Z 626.711,A -85,B 0,C 180,E1 -26918.167,E2 -26918.167} C_VEL
LIN {X 0,Y 246.389,Z 626.721,A -85,B 0,C 180,E1 -26923.145,E2 -26923.145} C_VEL
LIN {X 0,Y 246.254,Z 626.74,A -85,B 0,C 180,E1 -26926.525,E2 -26926.525} C_VEL
LIN {X 0,Y 246.255,Z 626.743,A -85,B 0,C 180,E1 -26930.177,E2 -26930.177} C_VEL
LIN {X 0,Y 246.197,Z 626.745,A -85,B 0,C 180,E1 -26934.439,E2 -26934.439} C_VEL
LIN {X 0,Y 246.126,Z 626.757,A -85,B 0,C 180,E1 -26938.934,E2 -26938.934} C_VEL
LIN {X 0,Y 246.151,Z 626.75,A -85,B 0,C 180,E1 -26942.728,E2 -26942.728} C_VEL
LIN {X 0,Y 246.178,Z 626.75,A -85,B 0,C 180,E1 -26947.187,E2 -26947.187} C_VEL
LIN {X 0,Y 246.141,Z 626.754,A -85,B 0,C 180,E1 -26950.882,E2 -26950.882} C_VEL
LIN {X 0,Y 246.124,Z 626.754,A -85,B 0,C 180,E1 -26955.355,E2 -26955.355} C_VEL
LIN {X 0,Y 246.14,Z 626.755,A -85,B 0,C 180,E1 -26959.118,E2 -26959.118} C_VEL
LIN {X 0,Y 246.164,Z 626.748,A -85,B 0,C 180,E1 -26963.307,E2 -26963.307} C_VEL
LIN {X 0,Y 246.116,Z 626.758,A -85,B 0,C 180,E1 -26967.267,E2 -26967.267} C_VEL
LIN {X 0,Y 246.163,Z 626.753,A -85,B 0,C 180,E1 -26971.895,E2 -26971.895} C_VEL
LIN {X 0,Y 246.183,Z 626.75,A -85,B 0,C 180,E1 -26976.527,E2 -26976.527} C_VEL
LIN {X 0,Y 246.258,Z 626.743,A -85,B 0,C 180,E1 -26980.043,E2 -26980.043} C_VEL
LIN {X 0,Y 246.337,Z 626.729,A -85,B 0,C 180,E1 -26985.187,E2 -26985.187} C_VEL
LIN {X 0,Y 246.437,Z 626.719,A -85,B 0,C 180,E1 -26990.182,E2 -26990.182} C_VEL
LIN {X 0,Y 246.75,Z 626.675,A -85,B 0,C 180,E1 -26993.481,E2 -26993.481} C_VEL
LIN {X 0,Y 246.767,Z 626.677,A -85,B 0,C 180,E1 -26996.746,E2 -26996.746} C_VEL
LIN {X 0,Y 246.906,Z 626.661,A -85,B 0,C 180,E1 -27000.001,E2 -27000.001} C_VEL
LIN {X 0,Y 246.697,Z 626.684,A -85,B 0,C 180,E1 -27004.887,E2 -27004.887} C_VEL
LIN {X 0,Y 246.52,Z 626.71,A -85,B 0,C 180,E1 -27008.168,E2 -27008.168} C_VEL
LIN {X 0,Y 246.342,Z 626.726,A -85,B 0,C 180,E1 -27013.149,E2 -27013.149} C_VEL
LIN {X 0,Y 246.219,Z 626.746,A -85,B 0,C 180,E1 -27016.528,E2 -27016.528} C_VEL
LIN {X 0,Y 246.191,Z 626.748,A -85,B 0,C 180,E1 -27020.134,E2 -27020.134} C_VEL
LIN {X 0,Y 246.2,Z 626.748,A -85,B 0,C 180,E1 -27024.439,E2 -27024.439} C_VEL
LIN {X 0,Y 246.121,Z 626.756,A -85,B 0,C 180,E1 -27028.935,E2 -27028.935} C_VEL
LIN {X 0,Y 246.11,Z 626.756,A -85,B 0,C 180,E1 -27032.735,E2 -27032.735} C_VEL
LIN {X 0,Y 246.102,Z 626.76,A -85,B 0,C 180,E1 -27037.163,E2 -27037.163} C_VEL
LIN {X 0,Y 246.09,Z 626.756,A -85,B 0,C 180,E1 -27040.893,E2 -27040.893} C_VEL
LIN {X 0,Y 246.072,Z 626.764,A -85,B 0,C 180,E1 -27045.368,E2 -27045.368} C_VEL
LIN {X 0,Y 246.115,Z 626.755,A -85,B 0,C 180,E1 -27050.213,E2 -27050.213} C_VEL
LIN {X 0,Y 246.103,Z 626.758,A -85,B 0,C 180,E1 -27053.296,E2 -27053.296} C_VEL
LIN {X 0,Y 246.109,Z 626.759,A -85,B 0,C 180,E1 -27057.265,E2 -27057.265} C_VEL
LIN {X 0,Y 246.241,Z 626.74,A -85,B 0,C 180,E1 -27061.862,E2 -27061.862} C_VEL
LIN {X 0,Y 246.454,Z 626.805,A -85,B 0,C 180,E1 -27063.409,E2 -27063.409} C_VEL
LIN {X 0,Y 247.811,Z 634.173,A -85,B 0,C 180,E1 -27066.289,E2 -27066.289} C_VEL
LIN {X 0,Y 246.621,Z 641.616,A -85,B 0,C 180,E1 -27069.059,E2 -27069.059} C_VEL
LIN {X 0,Y 247.205,Z 660.425,A -85,B 0,C 180,E1 -27069.95,E2 -27069.95} C_VEL
LIN {X 0,Y 249.607,Z 689.631,A -85,B 0,C 180,E1 -27071.333,E2 -27071.333} C_VEL
LIN {X 0,Y 248.04,Z 743.512,A -85,B 0,C 180,E1 -27073.856,E2 -27073.856} C_VEL
LIN {X 0,Y 247.362,Z 749.203,A -85,B 0,C 180,E1 -27074.163,E2 -27074.163} C_VEL
LIN {X 0,Y 244.052,Z 758.142,A -85,B 0,C 180,E1 -27074.802,E2 -27074.802} C_VEL
LIN {X 0,Y 240.536,Z 766.898,A -85,B 0,C 180,E1 -27075.595,E2 -27075.595} C_VEL
LIN {X 0,Y 239.736,Z 772.319,A -85,B 0,C 180,E1 -27076.16,E2 -27076.16} C_VEL
LIN {X 0,Y 239.068,Z 785.426,A -85,B 0,C 180,E1 -27077.736,E2 -27077.736} C_VEL
LIN {X 0,Y 238.428,Z 796.311,A -85,B 0,C 180,E1 -27079.42,E2 -27079.42} C_VEL
LIN {X 0,Y 237.947,Z 805.385,A -85,B 0,C 180,E1 -27081.11,E2 -27081.11} C_VEL
LIN {X 0,Y 237.575,Z 813.089,A -85,B 0,C 180,E1 -27082.802,E2 -27082.802} C_VEL
LIN {X 0,Y 237.359,Z 821.171,A -85,B 0,C 180,E1 -27084.921,E2 -27084.921} C_VEL
LIN {X 0,Y 237.209,Z 827.891,A -85,B 0,C 180,E1 -27087.038,E2 -27087.038} C_VEL
LIN {X 0,Y 237.077,Z 833.474,A -85,B 0,C 180,E1 -27089.154,E2 -27089.154} C_VEL
LIN {X 0,Y 236.87,Z 838.759,A -85,B 0,C 180,E1 -27091.695,E2 -27091.695} C_VEL
LIN {X 0,Y 236.546,Z 842.864,A -85,B 0,C 180,E1 -27094.246,E2 -27094.246} C_VEL
LIN {X 0,Y 236.504,Z 845.989,A -85,B 0,C 180,E1 -27096.804,E2 -27096.804} C_VEL
LIN {X 0,Y 237.411,Z 848.683,A -85,B 0,C 180,E1 -27100.197,E2 -27100.197} C_VEL
LIN {X 0,Y 238.261,Z 849.522,A -85,B 0,C 180,E1 -27101.876,E2 -27101.876} C_VEL
LIN {X 0,Y 240.664,Z 850.063,A -85,B 0,C 180,E1 -27105.186,E2 -27105.186} C_VEL
LIN {X 0,Y 244.106,Z 849.026,A -85,B 0,C 180,E1 -27108.4,E2 -27108.4} C_VEL
LIN {X 0,Y 246.129,Z 847.978,A -85,B 0,C 180,E1 -27109.969,E2 -27109.969} C_VEL
LIN {X 0,Y 250.966,Z 844.787,A -85,B 0,C 180,E1 -27113.001,E2 -27113.001} C_VEL
LIN {X 0,Y 256.71,Z 839.787,A -85,B 0,C 180,E1 -27115.885,E2 -27115.885} C_VEL
LIN {X 0,Y 261.529,Z 834.92,A -85,B 0,C 180,E1 -27117.95,E2 -27117.95} C_VEL
LIN {X 0,Y 266.799,Z 828.923,A -85,B 0,C 180,E1 -27119.922,E2 -27119.922} C_VEL
LIN {X 0,Y 271.794,Z 822.51,A -85,B 0,C 180,E1 -27121.595,E2 -27121.595} C_VEL
LIN {X 0,Y 277.093,Z 814.883,A -85,B 0,C 180,E1 -27123.171,E2 -27123.171} C_VEL
LIN {X 0,Y 281.796,Z 807.467,A -85,B 0,C 180,E1 -27124.436,E2 -27124.436} C_VEL
LIN {X 0,Y 286.813,Z 798.571,A -85,B 0,C 180,E1 -27125.667,E2 -27125.667} C_VEL
LIN {X 0,Y 292.059,Z 787.849,A -85,B 0,C 180,E1 -27126.84,E2 -27126.84} C_VEL
LIN {X 0,Y 296.337,Z 777.754,A -85,B 0,C 180,E1 -27127.706,E2 -27127.706} C_VEL
LIN {X 0,Y 300.046,Z 767.374,A -85,B 0,C 180,E1 -27128.43,E2 -27128.43} C_VEL
LIN {X 0,Y 302.701,Z 758.827,A -85,B 0,C 180,E1 -27128.924,E2 -27128.924} C_VEL
LIN {X 0,Y 305.773,Z 746.541,A -85,B 0,C 180,E1 -27129.479,E2 -27129.479} C_VEL
LIN {X 0,Y 309.203,Z 728.187,A -85,B 0,C 180,E1 -27130.177,E2 -27130.177} C_VEL
LIN {X 0,Y 307.663,Z 723.082,A -85,B 0,C 180,E1 -27131.788,E2 -27131.788} C_VEL
LIN {X 0,Y 306.607,Z 719.68,A -85,B 0,C 180,E1 -27133.189,E2 -27133.189} C_VEL
LIN {X 0,Y 305.479,Z 716.46,A -85,B 0,C 180,E1 -27134.875,E2 -27134.875} C_VEL
LIN {X 0,Y 304.32,Z 712.217,A -85,B 0,C 180,E1 -27138.322,E2 -27138.322} C_VEL
LIN {X 0,Y 304.095,Z 711.7,A -85,B 0,C 180,E1 -27139.838,E2 -27139.838} C_VEL
LIN {X 0,Y 304.501,Z 711.903,A -85,B 0,C 180,E1 -27142.59,E2 -27142.59} C_VEL
LIN {X 0,Y 306.159,Z 715.387,A -85,B 0,C 180,E1 -27146.113,E2 -27146.113} C_VEL
LIN {X 0,Y 307.745,Z 719.001,A -85,B 0,C 180,E1 -27148.107,E2 -27148.107} C_VEL
LIN {X 0,Y 309.358,Z 723.12,A -85,B 0,C 180,E1 -27149.76,E2 -27149.76} C_VEL
LIN {X 0,Y 309.71,Z 723.884,A -85,B 0,C 180,E1 -27150.062,E2 -27150.062} C_VEL
LIN {X 0,Y 305.595,Z 745.265,A -85,B 0,C 180,E1 -27150.871,E2 -27150.871} C_VEL
LIN {X 0,Y 301.768,Z 759.401,A -85,B 0,C 180,E1 -27151.615,E2 -27151.615} C_VEL
LIN {X 0,Y 298.114,Z 770.096,A -85,B 0,C 180,E1 -27152.351,E2 -27152.351} C_VEL
LIN {X 0,Y 294.051,Z 780.436,A -85,B 0,C 180,E1 -27153.281,E2 -27153.281} C_VEL
LIN {X 0,Y 290.02,Z 789.207,A -85,B 0,C 180,E1 -27154.232,E2 -27154.232} C_VEL
LIN {X 0,Y 285.548,Z 797.716,A -85,B 0,C 180,E1 -27155.354,E2 -27155.354} C_VEL
LIN {X 0,Y 280.214,Z 806.586,A -85,B 0,C 180,E1 -27156.815,E2 -27156.815} C_VEL
LIN {X 0,Y 275.177,Z 814.09,A -85,B 0,C 180,E1 -27158.34,E2 -27158.34} C_VEL
LIN {X 0,Y 270.396,Z 820.428,A -85,B 0,C 180,E1 -27159.926,E2 -27159.926} C_VEL
LIN {X 0,Y 265.777,Z 825.822,A -85,B 0,C 180,E1 -27161.581,E2 -27161.581} C_VEL
LIN {X 0,Y 260.663,Z 830.994,A -85,B 0,C 180,E1 -27163.611,E2 -27163.611} C_VEL
